LIN {X 0,Y 312.332,Z 608.768,A -85,B 0,C 180,E1 -15582.014,E2 -15582.014} C_VEL
LIN {X 0,Y 313.413,Z 600.363,A -85,B 0,C 180,E1 -15583.949,E2 -15583.949} C_VEL
LIN {X 0,Y 314.465,Z 591.676,A -85,B 0,C 180,E1 -15585.557,E2 -15585.557} C_VEL
LIN {X 0,Y 315.456,Z 582.123,A -85,B 0,C 180,E1 -15587.002,E2 -15587.002} C_VEL
LIN {X 0,Y 316.582,Z 571.707,A -85,B 0,C 180,E1 -15588.274,E2 -15588.274} C_VEL
LIN {X 0,Y 317.768,Z 560.291,A -85,B 0,C 180,E1 -15589.375,E2 -15589.375} C_VEL
LIN {X 0,Y 318.765,Z 548.571,A -85,B 0,C 180,E1 -15590.235,E2 -15590.235} C_VEL
LIN {X 0,Y 319.621,Z 535.041,A -85,B 0,C 180,E1 -15590.935,E2 -15590.935} C_VEL
LIN {X 0,Y 320.129,Z 521.595,A -85,B 0,C 180,E1 -15591.364,E2 -15591.364} C_VEL
LIN {X 0,Y 321.315,Z 456.274,A -85,B 0,C 180,E1 -15592.816,E2 -15592.816} C_VEL
LIN {X 0,Y 315.929,Z 420.388,A -85,B 0,C 180,E1 -15594.022,E2 -15594.022} C_VEL
LIN {X 0,Y 316.017,Z 418.253,A -85,B 0,C 180,E1 -15594.505,E2 -15594.505} C_VEL
LIN {X 0,Y 313.928,Z 406.505,A -85,B 0,C 180,E1 -15598.043,E2 -15598.043} C_VEL
LIN {X 0,Y 312.62,Z 400.101,A -85,B 0,C 180,E1 -15600.129,E2 -15600.129} C_VEL
LIN {X 0,Y 312.507,Z 400.053,A -85,B 0,C 180,E1 -15604.21,E2 -15604.21} C_VEL
LIN {X 0,Y 312.535,Z 400.049,A -85,B 0,C 180,E1 -15608.089,E2 -15608.089} C_VEL
LIN {X 0,Y 312.518,Z 400.054,A -85,B 0,C 180,E1 -15612.426,E2 -15612.426} C_VEL
LIN {X 0,Y 312.533,Z 400.041,A -85,B 0,C 180,E1 -15616.02,E2 -15616.02} C_VEL
LIN {X 0,Y 312.529,Z 400.055,A -85,B 0,C 180,E1 -15619.868,E2 -15619.868} C_VEL
LIN {X 0,Y 312.551,Z 400.049,A -85,B 0,C 180,E1 -15622.618,E2 -15622.618} C_VEL
LIN {X 0,Y 312.517,Z 400.054,A -85,B 0,C 180,E1 -15626.311,E2 -15626.311} C_VEL
LIN {X 0,Y 312.542,Z 400.047,A -85,B 0,C 180,E1 -15630.35,E2 -15630.35} C_VEL
LIN {X 0,Y 312.599,Z 400.044,A -85,B 0,C 180,E1 -15634.064,E2 -15634.064} C_VEL
LIN {X 0,Y 312.561,Z 400.049,A -85,B 0,C 180,E1 -15637.527,E2 -15637.527} C_VEL
LIN {X 0,Y 312.634,Z 400.04,A -85,B 0,C 180,E1 -15641.656,E2 -15641.656} C_VEL
LIN {X 0,Y 312.69,Z 400.034,A -85,B 0,C 180,E1 -15645.686,E2 -15645.686} C_VEL
LIN {X 0,Y 312.694,Z 400.027,A -85,B 0,C 180,E1 -15649.641,E2 -15649.641} C_VEL
LIN {X 0,Y 312.849,Z 400.01,A -85,B 0,C 180,E1 -15652.254,E2 -15652.254} C_VEL
LIN {X 0,Y 312.712,Z 400.031,A -85,B 0,C 180,E1 -15654.842,E2 -15654.842} C_VEL
LIN {X 0,Y 312.986,Z 399.993,A -85,B 0,C 180,E1 -15658.713,E2 -15658.713} C_VEL
LIN {X 0,Y 312.986,Z 399.99,A -85,B 0,C 180,E1 -15661.287,E2 -15661.287} C_VEL
LIN {X 0,Y 312.712,Z 400.032,A -85,B 0,C 180,E1 -15665.158,E2 -15665.158} C_VEL
LIN {X 0,Y 312.849,Z 400.013,A -85,B 0,C 180,E1 -15667.746,E2 -15667.746} C_VEL
LIN {X 0,Y 312.664,Z 400.027,A -85,B 0,C 180,E1 -15671.671,E2 -15671.671} C_VEL
LIN {X 0,Y 312.696,Z 400.029,A -85,B 0,C 180,E1 -15674.887,E2 -15674.887} C_VEL
LIN {X 0,Y 312.627,Z 400.044,A -85,B 0,C 180,E1 -15679.237,E2 -15679.237} C_VEL
LIN {X 0,Y 312.542,Z 400.047,A -85,B 0,C 180,E1 -15682.789,E2 -15682.789} C_VEL
LIN {X 0,Y 312.599,Z 400.041,A -85,B 0,C 180,E1 -15685.936,E2 -15685.936} C_VEL
LIN {X 0,Y 312.542,Z 400.051,A -85,B 0,C 180,E1 -15689.65,E2 -15689.65} C_VEL
LIN {X 0,Y 312.516,Z 400.048,A -85,B 0,C 180,E1 -15693.689,E2 -15693.689} C_VEL
LIN {X 0,Y 312.518,Z 400.057,A -85,B 0,C 180,E1 -15697.386,E2 -15697.386} C_VEL
LIN {X 0,Y 312.488,Z 400.058,A -85,B 0,C 180,E1 -15700.709,E2 -15700.709} C_VEL
LIN {X 0,Y 312.472,Z 400.058,A -85,B 0,C 180,E1 -15704.206,E2 -15704.206} C_VEL
LIN {X 0,Y 312.527,Z 400.05,A -85,B 0,C 180,E1 -15707.91,E2 -15707.91} C_VEL
LIN {X 0,Y 312.542,Z 400.052,A -85,B 0,C 180,E1 -15711.909,E2 -15711.909} C_VEL
LIN {X 0,Y 312.506,Z 400.048,A -85,B 0,C 180,E1 -15715.79,E2 -15715.79} C_VEL
LIN {X 0,Y 312.523,Z 400.047,A -85,B 0,C 180,E1 -15718.854,E2 -15718.854} C_VEL
LIN {X 0,Y 312.574,Z 400.047,A -85,B 0,C 180,E1 -15721.825,E2 -15721.825} C_VEL
LIN {X 0,Y 312.586,Z 400.042,A -85,B 0,C 180,E1 -15724.711,E2 -15724.711} C_VEL
LIN {X 0,Y 312.588,Z 400.047,A -85,B 0,C 180,E1 -15727.529,E2 -15727.529} C_VEL
LIN {X 0,Y 312.639,Z 400.028,A -85,B 0,C 180,E1 -15731.656,E2 -15731.656} C_VEL
LIN {X 0,Y 312.701,Z 400.206,A -85,B 0,C 180,E1 -15735.147,E2 -15735.147} C_VEL
LIN {X 0,Y 314.592,Z 410.211,A -85,B 0,C 180,E1 -15738.401,E2 -15738.401} C_VEL
LIN {X 0,Y 314.972,Z 412.171,A -85,B 0,C 180,E1 -15738.949,E2 -15738.949} C_VEL
LIN {X 0,Y 317.49,Z 420.363,A -85,B 0,C 180,E1 -15739.351,E2 -15739.351} C_VEL
LIN {X 0,Y 320.696,Z 439.395,A -85,B 0,C 180,E1 -15740.005,E2 -15740.005} C_VEL
LIN {X 0,Y 321.593,Z 445.108,A -85,B 0,C 180,E1 -15740.193,E2 -15740.193} C_VEL
LIN {X 0,Y 319.963,Z 519.638,A -85,B 0,C 180,E1 -15741.871,E2 -15741.871} C_VEL
LIN {X 0,Y 319.365,Z 532.672,A -85,B 0,C 180,E1 -15742.413,E2 -15742.413} C_VEL
LIN {X 0,Y 318.56,Z 545.103,A -85,B 0,C 180,E1 -15743.177,E2 -15743.177} C_VEL
LIN {X 0,Y 317.505,Z 556.543,A -85,B 0,C 180,E1 -15744.124,E2 -15744.124} C_VEL
LIN {X 0,Y 316.221,Z 568.185,A -85,B 0,C 180,E1 -15745.379,E2 -15745.379} C_VEL
LIN {X 0,Y 314.984,Z 578.646,A -85,B 0,C 180,E1 -15746.802,E2 -15746.802} C_VEL
LIN {X 0,Y 313.883,Z 588.052,A -85,B 0,C 180,E1 -15748.396,E2 -15748.396} C_VEL
LIN {X 0,Y 312.774,Z 597.128,A -85,B 0,C 180,E1 -15750.322,E2 -15750.322} C_VEL
LIN {X 0,Y 312.008,Z 604.437,A -85,B 0,C 180,E1 -15752.259,E2 -15752.259} C_VEL
LIN {X 0,Y 311.384,Z 609.404,A -85,B 0,C 180,E1 -15753.882,E2 -15753.882} C_VEL
LIN {X 0,Y 311.069,Z 614.19,A -85,B 0,C 180,E1 -15755.827,E2 -15755.827} C_VEL
LIN {X 0,Y 310.787,Z 617.906,A -85,B 0,C 180,E1 -15757.798,E2 -15757.798} C_VEL
LIN {X 0,Y 310.591,Z 619.823,A -85,B 0,C 180,E1 -15759.113,E2 -15759.113} C_VEL
LIN {X 0,Y 310.484,Z 621.266,A -85,B 0,C 180,E1 -15760.432,E2 -15760.432} C_VEL
LIN {X 0,Y 310.487,Z 622.287,A -85,B 0,C 180,E1 -15761.754,E2 -15761.754} C_VEL
LIN {X 0,Y 310.52,Z 622.988,A -85,B 0,C 180,E1 -15763.29,E2 -15763.29} C_VEL
LIN {X 0,Y 310.477,Z 622.899,A -85,B 0,C 180,E1 -15765.761,E2 -15765.761} C_VEL
LIN {X 0,Y 310.849,Z 621.362,A -85,B 0,C 180,E1 -15768.272,E2 -15768.272} C_VEL
LIN {X 0,Y 311.123,Z 619.69,A -85,B 0,C 180,E1 -15769.805,E2 -15769.805} C_VEL
LIN {X 0,Y 311.721,Z 616.547,A -85,B 0,C 180,E1 -15771.839,E2 -15771.839} C_VEL
LIN {X 0,Y 312.536,Z 612.255,A -85,B 0,C 180,E1 -15773.876,E2 -15773.876} C_VEL
LIN {X 0,Y 313.634,Z 606.844,A -85,B 0,C 180,E1 -15775.854,E2 -15775.854} C_VEL
LIN {X 0,Y 315.1,Z 599.633,A -85,B 0,C 180,E1 -15777.929,E2 -15777.929} C_VEL
LIN {X 0,Y 316.754,Z 591.555,A -85,B 0,C 180,E1 -15779.771,E2 -15779.771} C_VEL
LIN {X 0,Y 318.433,Z 582.51,A -85,B 0,C 180,E1 -15781.426,E2 -15781.426} C_VEL
LIN {X 0,Y 320.298,Z 572.505,A -85,B 0,C 180,E1 -15782.891,E2 -15782.891} C_VEL
LIN {X 0,Y 321.96,Z 561.76,A -85,B 0,C 180,E1 -15784.159,E2 -15784.159} C_VEL
LIN {X 0,Y 323.509,Z 549.927,A -85,B 0,C 180,E1 -15785.242,E2 -15785.242} C_VEL
LIN {X 0,Y 324.743,Z 538.352,A -85,B 0,C 180,E1 -15786.041,E2 -15786.041} C_VEL
LIN {X 0,Y 325.821,Z 525.426,A -85,B 0,C 180,E1 -15786.67,E2 -15786.67} C_VEL
LIN {X 0,Y 326.468,Z 511.967,A -85,B 0,C 180,E1 -15787.067,E2 -15787.067} C_VEL
LIN {X 0,Y 328.157,Z 446.992,A -85,B 0,C 180,E1 -15788.521,E2 -15788.521} C_VEL
LIN {X 0,Y 325.249,Z 434.051,A -85,B 0,C 180,E1 -15789.147,E2 -15789.147} C_VEL
LIN {X 0,Y 321.952,Z 426.371,A -85,B 0,C 180,E1 -15789.693,E2 -15789.693} C_VEL
LIN {X 0,Y 319.927,Z 423.383,A -85,B 0,C 180,E1 -15789.995,E2 -15789.995} C_VEL
LIN {X 0,Y 315.274,Z 419.81,A -85,B 0,C 180,E1 -15790.605,E2 -15790.605} C_VEL
LIN {X 0,Y 310.624,Z 416.297,A -85,B 0,C 180,E1 -15791.239,E2 -15791.239} C_VEL
LIN {X 0,Y 308.623,Z 413.402,A -85,B 0,C 180,E1 -15791.58,E2 -15791.58} C_VEL
LIN {X 0,Y 308.228,Z 412.248,A -85,B 0,C 180,E1 -15791.753,E2 -15791.753} C_VEL
LIN {X 0,Y 306.422,Z 404.582,A -85,B 0,C 180,E1 -15794.683,E2 -15794.683} C_VEL
LIN {X 0,Y 305.53,Z 400.961,A -85,B 0,C 180,E1 -15796.243,E2 -15796.243} C_VEL
LIN {X 0,Y 305.48,Z 400.933,A -85,B 0,C 180,E1 -15799.896,E2 -15799.896} C_VEL
LIN {X 0,Y 305.496,Z 400.931,A -85,B 0,C 180,E1 -15803.626,E2 -15803.626} C_VEL
LIN {X 0,Y 305.46,Z 400.927,A -85,B 0,C 180,E1 -15806.483,E2 -15806.483} C_VEL
LIN {X 0,Y 305.46,Z 400.916,A -85,B 0,C 180,E1 -15809.591,E2 -15809.591} C_VEL
LIN {X 0,Y 305.528,Z 400.927,A -85,B 0,C 180,E1 -15812.609,E2 -15812.609} C_VEL
LIN {X 0,Y 305.502,Z 400.93,A -85,B 0,C 180,E1 -15815.538,E2 -15815.538} C_VEL
LIN {X 0,Y 305.524,Z 400.927,A -85,B 0,C 180,E1 -15819.815,E2 -15819.815} C_VEL
LIN {X 0,Y 305.568,Z 400.918,A -85,B 0,C 180,E1 -15822.603,E2 -15822.603} C_VEL
LIN {X 0,Y 305.642,Z 400.904,A -85,B 0,C 180,E1 -15825.349,E2 -15825.349} C_VEL
LIN {X 0,Y 305.633,Z 400.903,A -85,B 0,C 180,E1 -15829.4,E2 -15829.4} C_VEL
LIN {X 0,Y 305.805,Z 400.892,A -85,B 0,C 180,E1 -15832.074,E2 -15832.074} C_VEL
LIN {X 0,Y 305.686,Z 400.897,A -85,B 0,C 180,E1 -15834.724,E2 -15834.724} C_VEL
LIN {X 0,Y 305.955,Z 400.864,A -85,B 0,C 180,E1 -15838.684,E2 -15838.684} C_VEL
LIN {X 0,Y 305.954,Z 400.874,A -85,B 0,C 180,E1 -15841.316,E2 -15841.316} C_VEL
LIN {X 0,Y 305.684,Z 400.905,A -85,B 0,C 180,E1 -15845.277,E2 -15845.277} C_VEL
LIN {X 0,Y 305.805,Z 400.886,A -85,B 0,C 180,E1 -15847.926,E2 -15847.926} C_VEL
LIN {X 0,Y 305.599,Z 400.917,A -85,B 0,C 180,E1 -15851.945,E2 -15851.945} C_VEL
LIN {X 0,Y 305.631,Z 400.911,A -85,B 0,C 180,E1 -15855.035,E2 -15855.035} C_VEL
LIN {X 0,Y 305.57,Z 400.919,A -85,B 0,C 180,E1 -15859.446,E2 -15859.446} C_VEL
LIN {X 0,Y 305.484,Z 400.924,A -85,B 0,C 180,E1 -15863.042,E2 -15863.042} C_VEL
LIN {X 0,Y 305.541,Z 400.919,A -85,B 0,C 180,E1 -15866.228,E2 -15866.228} C_VEL
LIN {X 0,Y 305.49,Z 400.931,A -85,B 0,C 180,E1 -15869.051,E2 -15869.051} C_VEL
LIN {X 0,Y 305.46,Z 400.932,A -85,B 0,C 180,E1 -15873.518,E2 -15873.518} C_VEL
LIN {X 0,Y 305.498,Z 400.927,A -85,B 0,C 180,E1 -15876.736,E2 -15876.736} C_VEL
LIN {X 0,Y 305.49,Z 400.914,A -85,B 0,C 180,E1 -15880.609,E2 -15880.609} C_VEL
LIN {X 0,Y 305.489,Z 400.932,A -85,B 0,C 180,E1 -15883.644,E2 -15883.644} C_VEL
LIN {X 0,Y 305.48,Z 400.925,A -85,B 0,C 180,E1 -15887.41,E2 -15887.41} C_VEL
LIN {X 0,Y 305.493,Z 400.932,A -85,B 0,C 180,E1 -15891.602,E2 -15891.602} C_VEL
LIN {X 0,Y 305.498,Z 401.029,A -85,B 0,C 180,E1 -15894.691,E2 -15894.691} C_VEL
LIN {X 0,Y 307.861,Z 410.376,A -85,B 0,C 180,E1 -15898.329,E2 -15898.329} C_VEL
LIN {X 0,Y 309.922,Z 419.562,A -85,B 0,C 180,E1 -15901.563,E2 -15901.563} C_VEL
LIN {X 0,Y 313.421,Z 427.22,A -85,B 0,C 180,E1 -15902.233,E2 -15902.233} C_VEL
LIN {X 0,Y 316.75,Z 435.265,A -85,B 0,C 180,E1 -15902.823,E2 -15902.823} C_VEL
LIN {X 0,Y 320.789,Z 454.521,A -85,B 0,C 180,E1 -15903.763,E2 -15903.763} C_VEL
LIN {X 0,Y 321.79,Z 460.542,A -85,B 0,C 180,E1 -15904.023,E2 -15904.023} C_VEL
LIN {X 0,Y 319.782,Z 527.928,A -85,B 0,C 180,E1 -15905.579,E2 -15905.579} C_VEL
LIN {X 0,Y 318.81,Z 540.907,A -85,B 0,C 180,E1 -15906.106,E2 -15906.106} C_VEL
LIN {X 0,Y 317.437,Z 553.468,A -85,B 0,C 180,E1 -15906.861,E2 -15906.861} C_VEL
LIN {X 0,Y 316.006,Z 564.655,A -85,B 0,C 180,E1 -15907.786,E2 -15907.786} C_VEL
LIN {X 0,Y 314.12,Z 576.238,A -85,B 0,C 180,E1 -15909.025,E2 -15909.025} C_VEL
LIN {X 0,Y 312.255,Z 586.659,A -85,B 0,C 180,E1 -15910.441,E2 -15910.441} C_VEL
LIN {X 0,Y 310.511,Z 595.458,A -85,B 0,C 180,E1 -15911.919,E2 -15911.919} C_VEL
LIN {X 0,Y 308.774,Z 604.486,A -85,B 0,C 180,E1 -15913.811,E2 -15913.811} C_VEL
LIN {X 0,Y 307.072,Z 611.943,A -85,B 0,C 180,E1 -15915.758,E2 -15915.758} C_VEL
LIN {X 0,Y 305.684,Z 618.85,A -85,B 0,C 180,E1 -15918.059,E2 -15918.059} C_VEL
LIN {X 0,Y 304.772,Z 623.43,A -85,B 0,C 180,E1 -15920.041,E2 -15920.041} C_VEL
LIN {X 0,Y 304.128,Z 626.927,A -85,B 0,C 180,E1 -15922.031,E2 -15922.031} C_VEL
LIN {X 0,Y 303.783,Z 629.584,A -85,B 0,C 180,E1 -15924.159,E2 -15924.159} C_VEL
LIN {X 0,Y 303.608,Z 631.026,A -85,B 0,C 180,E1 -15926.018,E2 -15926.018} C_VEL
LIN {X 0,Y 303.582,Z 631.609,A -85,B 0,C 180,E1 -15927.347,E2 -15927.347} C_VEL
LIN {X 0,Y 303.528,Z 631.779,A -85,B 0,C 180,E1 -15928.674,E2 -15928.674} C_VEL
LIN {X 0,Y 303.545,Z 631.537,A -85,B 0,C 180,E1 -15930,E2 -15930} C_VEL
LIN {X 0,Y 303.58,Z 629.892,A -85,B 0,C 180,E1 -15932.654,E2 -15932.654} C_VEL
LIN {X 0,Y 303.584,Z 628.446,A -85,B 0,C 180,E1 -15933.983,E2 -15933.983} C_VEL
LIN {X 0,Y 303.618,Z 626.19,A -85,B 0,C 180,E1 -15935.53,E2 -15935.53} C_VEL
LIN {X 0,Y 303.995,Z 621.397,A -85,B 0,C 180,E1 -15937.974,E2 -15937.974} C_VEL
LIN {X 0,Y 304.608,Z 615.141,A -85,B 0,C 180,E1 -15940.301,E2 -15940.301} C_VEL
LIN {X 0,Y 305.353,Z 608.311,A -85,B 0,C 180,E1 -15942.292,E2 -15942.292} C_VEL
LIN {X 0,Y 306.473,Z 599.799,A -85,B 0,C 180,E1 -15944.272,E2 -15944.272} C_VEL
LIN {X 0,Y 307.726,Z 589.82,A -85,B 0,C 180,E1 -15946.111,E2 -15946.111} C_VEL
LIN {X 0,Y 308.901,Z 578.948,A -85,B 0,C 180,E1 -15947.716,E2 -15947.716} C_VEL
LIN {X 0,Y 310.122,Z 567.713,A -85,B 0,C 180,E1 -15949.012,E2 -15949.012} C_VEL
LIN {X 0,Y 311.398,Z 555.107,A -85,B 0,C 180,E1 -15950.132,E2 -15950.132} C_VEL
LIN {X 0,Y 312.406,Z 542.157,A -85,B 0,C 180,E1 -15950.967,E2 -15950.967} C_VEL
LIN {X 0,Y 313.17,Z 528.284,A -85,B 0,C 180,E1 -15951.56,E2 -15951.56} C_VEL
LIN {X 0,Y 314.635,Z 457.597,A -85,B 0,C 180,E1 -15953.196,E2 -15953.196} C_VEL
LIN {X 0,Y 309.07,Z 420.436,A -85,B 0,C 180,E1 -15954.474,E2 -15954.474} C_VEL
LIN {X 0,Y 309.035,Z 419.339,A -85,B 0,C 180,E1 -15954.659,E2 -15954.659} C_VEL
LIN {X 0,Y 307.124,Z 408.508,A -85,B 0,C 180,E1 -15957.976,E2 -15957.976} C_VEL
LIN {X 0,Y 305.525,Z 401.019,A -85,B 0,C 180,E1 -15960.45,E2 -15960.45} C_VEL
LIN {X 0,Y 305.465,Z 400.931,A -85,B 0,C 180,E1 -15964.078,E2 -15964.078} C_VEL
LIN {X 0,Y 305.496,Z 400.93,A -85,B 0,C 180,E1 -15966.736,E2 -15966.736} C_VEL
LIN {X 0,Y 305.454,Z 400.933,A -85,B 0,C 180,E1 -15970.599,E2 -15970.599} C_VEL
LIN {X 0,Y 305.452,Z 400.931,A -85,B 0,C 180,E1 -15973.65,E2 -15973.65} C_VEL
LIN {X 0,Y 305.506,Z 400.918,A -85,B 0,C 180,E1 -15977.403,E2 -15977.403} C_VEL
LIN {X 0,Y 305.518,Z 400.929,A -85,B 0,C 180,E1 -15981.604,E2 -15981.604} C_VEL
LIN {X 0,Y 305.46,Z 400.93,A -85,B 0,C 180,E1 -15984.886,E2 -15984.886} C_VEL
LIN {X 0,Y 305.449,Z 400.935,A -85,B 0,C 180,E1 -15988.355,E2 -15988.355} C_VEL
LIN {X 0,Y 305.518,Z 400.924,A -85,B 0,C 180,E1 -15991.113,E2 -15991.113} C_VEL
LIN {X 0,Y 305.568,Z 400.92,A -85,B 0,C 180,E1 -15994.087,E2 -15994.087} C_VEL
LIN {X 0,Y 305.478,Z 400.926,A -85,B 0,C 180,E1 -15998.401,E2 -15998.401} C_VEL
LIN {X 0,Y 305.576,Z 400.915,A -85,B 0,C 180,E1 -16001.217,E2 -16001.217} C_VEL
LIN {X 0,Y 305.645,Z 400.914,A -85,B 0,C 180,E1 -16005.349,E2 -16005.349} C_VEL
LIN {X 0,Y 305.631,Z 400.905,A -85,B 0,C 180,E1 -16009.399,E2 -16009.399} C_VEL
LIN {X 0,Y 305.793,Z 400.889,A -85,B 0,C 180,E1 -16012.074,E2 -16012.074} C_VEL
LIN {X 0,Y 305.683,Z 400.906,A -85,B 0,C 180,E1 -16014.723,E2 -16014.723} C_VEL
LIN {X 0,Y 305.953,Z 400.869,A -85,B 0,C 180,E1 -16018.684,E2 -16018.684} C_VEL
LIN {X 0,Y 305.953,Z 400.865,A -85,B 0,C 180,E1 -16021.316,E2 -16021.316} C_VEL
LIN {X 0,Y 305.683,Z 400.909,A -85,B 0,C 180,E1 -16025.277,E2 -16025.277} C_VEL
LIN {X 0,Y 305.793,Z 400.891,A -85,B 0,C 180,E1 -16027.926,E2 -16027.926} C_VEL
LIN {X 0,Y 305.598,Z 400.905,A -85,B 0,C 180,E1 -16031.945,E2 -16031.945} C_VEL
LIN {X 0,Y 305.634,Z 400.909,A -85,B 0,C 180,E1 -16035.035,E2 -16035.035} C_VEL
LIN {X 0,Y 305.573,Z 400.92,A -85,B 0,C 180,E1 -16039.445,E2 -16039.445} C_VEL
LIN {X 0,Y 305.487,Z 400.924,A -85,B 0,C 180,E1 -16043.041,E2 -16043.041} C_VEL
LIN {X 0,Y 305.544,Z 400.919,A -85,B 0,C 180,E1 -16046.227,E2 -16046.227} C_VEL
LIN {X 0,Y 305.493,Z 400.933,A -85,B 0,C 180,E1 -16049.05,E2 -16049.05} C_VEL
LIN {X 0,Y 305.462,Z 400.927,A -85,B 0,C 180,E1 -16053.517,E2 -16053.517} C_VEL
LIN {X 0,Y 305.47,Z 400.932,A -85,B 0,C 180,E1 -16056.74,E2 -16056.74} C_VEL
LIN {X 0,Y 305.452,Z 400.933,A -85,B 0,C 180,E1 -16060.6,E2 -16060.6} C_VEL
LIN {X 0,Y 305.423,Z 400.937,A -85,B 0,C 180,E1 -16064.494,E2 -16064.494} C_VEL
LIN {X 0,Y 305.475,Z 400.929,A -85,B 0,C 180,E1 -16068.15,E2 -16068.15} C_VEL
LIN {X 0,Y 305.507,Z 400.929,A -85,B 0,C 180,E1 -16071.603,E2 -16071.603} C_VEL
LIN {X 0,Y 305.462,Z 400.931,A -85,B 0,C 180,E1 -16074.887,E2 -16074.887} C_VEL
LIN {X 0,Y 305.451,Z 400.923,A -85,B 0,C 180,E1 -16078.355,E2 -16078.355} C_VEL
LIN {X 0,Y 305.52,Z 400.93,A -85,B 0,C 180,E1 -16081.114,E2 -16081.114} C_VEL
LIN {X 0,Y 305.566,Z 400.915,A -85,B 0,C 180,E1 -16084.088,E2 -16084.088} C_VEL
LIN {X 0,Y 305.502,Z 400.93,A -85,B 0,C 180,E1 -16088.403,E2 -16088.403} C_VEL
LIN {X 0,Y 305.591,Z 400.904,A -85,B 0,C 180,E1 -16091.218,E2 -16091.218} C_VEL
LIN {X 0,Y 305.658,Z 401.072,A -85,B 0,C 180,E1 -16094.813,E2 -16094.813} C_VEL
LIN {X 0,Y 307.557,Z 411.003,A -85,B 0,C 180,E1 -16098.132,E2 -16098.132} C_VEL
LIN {X 0,Y 307.829,Z 412.394,A -85,B 0,C 180,E1 -16098.479,E2 -16098.479} C_VEL
LIN {X 0,Y 310.923,Z 422.04,A -85,B 0,C 180,E1 -16098.96,E2 -16098.96} C_VEL
LIN {X 0,Y 314.103,Z 440.853,A -85,B 0,C 180,E1 -16099.623,E2 -16099.623} C_VEL
LIN {X 0,Y 314.893,Z 446.011,A -85,B 0,C 180,E1 -16099.797,E2 -16099.797} C_VEL
LIN {X 0,Y 313.253,Z 518.575,A -85,B 0,C 180,E1 -16101.452,E2 -16101.452} C_VEL
LIN {X 0,Y 312.698,Z 531.262,A -85,B 0,C 180,E1 -16101.965,E2 -16101.965} C_VEL
LIN {X 0,Y 311.83,Z 544.047,A -85,B 0,C 180,E1 -16102.741,E2 -16102.741} C_VEL
LIN {X 0,Y 310.79,Z 555.378,A -85,B 0,C 180,E1 -16103.671,E2 -16103.671} C_VEL
LIN {X 0,Y 309.594,Z 566.023,A -85,B 0,C 180,E1 -16104.79,E2 -16104.79} C_VEL
LIN {X 0,Y 308.478,Z 575.797,A -85,B 0,C 180,E1 -16106.081,E2 -16106.081} C_VEL
LIN {X 0,Y 307.176,Z 585.738,A -85,B 0,C 180,E1 -16107.705,E2 -16107.705} C_VEL
LIN {X 0,Y 306.254,Z 593.861,A -85,B 0,C 180,E1 -16109.342,E2 -16109.342} C_VEL
LIN {X 0,Y 305.197,Z 601.864,A -85,B 0,C 180,E1 -16111.319,E2 -16111.319} C_VEL
LIN {X 0,Y 304.475,Z 608.254,A -85,B 0,C 180,E1 -16113.308,E2 -16113.308} C_VEL
LIN {X 0,Y 304.063,Z 613.325,A -85,B 0,C 180,E1 -16115.304,E2 -16115.304} C_VEL
LIN {X 0,Y 303.777,Z 617.265,A -85,B 0,C 180,E1 -16117.31,E2 -16117.31} C_VEL
LIN {X 0,Y 303.473,Z 620.176,A -85,B 0,C 180,E1 -16119.329,E2 -16119.329} C_VEL
LIN {X 0,Y 303.384,Z 621.548,A -85,B 0,C 180,E1 -16120.679,E2 -16120.679} C_VEL
LIN {X 0,Y 303.383,Z 622.518,A -85,B 0,C 180,E1 -16122.033,E2 -16122.033} C_VEL
LIN {X 0,Y 303.427,Z 623.09,A -85,B 0,C 180,E1 -16123.392,E2 -16123.392} C_VEL
LIN {X 0,Y 303.361,Z 623.213,A -85,B 0,C 180,E1 -16124.763,E2 -16124.763} C_VEL
LIN {X 0,Y 303.408,Z 622.923,A -85,B 0,C 180,E1 -16126.138,E2 -16126.138} C_VEL
LIN {X 0,Y 303.81,Z 621.473,A -85,B 0,C 180,E1 -16128.478,E2 -16128.478} C_VEL
LIN {X 0,Y 304.357,Z 618.557,A -85,B 0,C 180,E1 -16130.971,E2 -16130.971} C_VEL
LIN {X 0,Y 305.095,Z 614.922,A -85,B 0,C 180,E1 -16133.053,E2 -16133.053} C_VEL
LIN {X 0,Y 306.123,Z 610.082,A -85,B 0,C 180,E1 -16135.132,E2 -16135.132} C_VEL
LIN {X 0,Y 307.444,Z 603.879,A -85,B 0,C 180,E1 -16137.205,E2 -16137.205} C_VEL
LIN {X 0,Y 309.108,Z 596.084,A -85,B 0,C 180,E1 -16139.263,E2 -16139.263} C_VEL
LIN {X 0,Y 310.946,Z 587.398,A -85,B 0,C 180,E1 -16141.079,E2 -16141.079} C_VEL
LIN {X 0,Y 312.756,Z 578.142,A -85,B 0,C 180,E1 -16142.635,E2 -16142.635} C_VEL
LIN {X 0,Y 314.492,Z 568.389,A -85,B 0,C 180,E1 -16143.963,E2 -16143.963} C_VEL
LIN {X 0,Y 316.152,Z 557.714,A -85,B 0,C 180,E1 -16145.129,E2 -16145.129} C_VEL
LIN {X 0,Y 317.704,Z 545.272,A -85,B 0,C 180,E1 -16146.181,E2 -16146.181} C_VEL
LIN {X 0,Y 319.049,Z 532.166,A -85,B 0,C 180,E1 -16146.968,E2 -16146.968} C_VEL
LIN {X 0,Y 319.913,Z 519.714,A -85,B 0,C 180,E1 -16147.471,E2 -16147.471} C_VEL
LIN {X 0,Y 322.056,Z 448.446,A -85,B 0,C 180,E1 -16149.111,E2 -16149.111} C_VEL
LIN {X 0,Y 319.404,Z 436.749,A -85,B 0,C 180,E1 -16149.698,E2 -16149.698} C_VEL
LIN {X 0,Y 312.065,Z 420.297,A -85,B 0,C 180,E1 -16150.961,E2 -16150.961} C_VEL
LIN {X 0,Y 308.623,Z 413.402,A -85,B 0,C 180,E1 -16151.58,E2 -16151.58} C_VEL
LIN {X 0,Y 307.63,Z 412.085,A -85,B 0,C 180,E1 -16151.882,E2 -16151.882} C_VEL
LIN {X 0,Y 302.646,Z 408.369,A -85,B 0,C 180,E1 -16153.836,E2 -16153.836} C_VEL
LIN {X 0,Y 300.585,Z 406.45,A -85,B 0,C 180,E1 -16154.954,E2 -16154.954} C_VEL
LIN {X 0,Y 299.117,Z 403.891,A -85,B 0,C 180,E1 -16156.07,E2 -16156.07} C_VEL
LIN {X 0,Y 298.534,Z 402.112,A -85,B 0,C 180,E1 -16156.826,E2 -16156.826} C_VEL
LIN {X 0,Y 298.47,Z 401.799,A -85,B 0,C 180,E1 -16157.393,E2 -16157.393} C_VEL
LIN {X 0,Y 298.431,Z 401.8,A -85,B 0,C 180,E1 -16160.998,E2 -16160.998} C_VEL
LIN {X 0,Y 298.428,Z 401.807,A -85,B 0,C 180,E1 -16163.932,E2 -16163.932} C_VEL
LIN {X 0,Y 298.394,Z 401.816,A -85,B 0,C 180,E1 -16167.981,E2 -16167.981} C_VEL
LIN {X 0,Y 298.464,Z 401.799,A -85,B 0,C 180,E1 -16171.904,E2 -16171.904} C_VEL
LIN {X 0,Y 298.48,Z 401.801,A -85,B 0,C 180,E1 -16174.924,E2 -16174.924} C_VEL
LIN {X 0,Y 298.451,Z 401.81,A -85,B 0,C 180,E1 -16179.315,E2 -16179.315} C_VEL
LIN {X 0,Y 298.532,Z 401.792,A -85,B 0,C 180,E1 -16182.179,E2 -16182.179} C_VEL
LIN {X 0,Y 298.586,Z 401.784,A -85,B 0,C 180,E1 -16184.994,E2 -16184.994} C_VEL
LIN {X 0,Y 298.588,Z 401.782,A -85,B 0,C 180,E1 -16189.147,E2 -16189.147} C_VEL
LIN {X 0,Y 298.751,Z 401.771,A -85,B 0,C 180,E1 -16191.886,E2 -16191.886} C_VEL
LIN {X 0,Y 298.657,Z 401.772,A -85,B 0,C 180,E1 -16194.599,E2 -16194.599} C_VEL
LIN {X 0,Y 298.922,Z 401.74,A -85,B 0,C 180,E1 -16198.653,E2 -16198.653} C_VEL
LIN {X 0,Y 298.92,Z 401.75,A -85,B 0,C 180,E1 -16201.347,E2 -16201.347} C_VEL
LIN {X 0,Y 298.654,Z 401.782,A -85,B 0,C 180,E1 -16205.401,E2 -16205.401} C_VEL
LIN {X 0,Y 298.751,Z 401.763,A -85,B 0,C 180,E1 -16208.114,E2 -16208.114} C_VEL
LIN {X 0,Y 298.549,Z 401.794,A -85,B 0,C 180,E1 -16212.232,E2 -16212.232} C_VEL
LIN {X 0,Y 298.599,Z 401.79,A -85,B 0,C 180,E1 -16215.21,E2 -16215.21} C_VEL
LIN {X 0,Y 298.533,Z 401.793,A -85,B 0,C 180,E1 -16219.244,E2 -16219.244} C_VEL
LIN {X 0,Y 298.451,Z 401.804,A -85,B 0,C 180,E1 -16223.598,E2 -16223.598} C_VEL
LIN {X 0,Y 298.484,Z 401.797,A -85,B 0,C 180,E1 -16226.575,E2 -16226.575} C_VEL
LIN {X 0,Y 298.415,Z 401.811,A -85,B 0,C 180,E1 -16229.642,E2 -16229.642} C_VEL
LIN {X 0,Y 298.39,Z 401.816,A -85,B 0,C 180,E1 -16232.801,E2 -16232.801} C_VEL
LIN {X 0,Y 298.466,Z 401.803,A -85,B 0,C 180,E1 -16236.815,E2 -16236.815} C_VEL
LIN {X 0,Y 298.451,Z 401.787,A -85,B 0,C 180,E1 -16241.104,E2 -16241.104} C_VEL
LIN {X 0,Y 298.456,Z 401.799,A -85,B 0,C 180,E1 -16243.117,E2 -16243.117} C_VEL
LIN {X 0,Y 298.429,Z 401.798,A -85,B 0,C 180,E1 -16246.927,E2 -16246.927} C_VEL
LIN {X 0,Y 298.413,Z 401.805,A -85,B 0,C 180,E1 -16251.004,E2 -16251.004} C_VEL
LIN {X 0,Y 298.476,Z 401.931,A -85,B 0,C 180,E1 -16253.94,E2 -16253.94} C_VEL
LIN {X 0,Y 300.951,Z 411.844,A -85,B 0,C 180,E1 -16257.91,E2 -16257.91} C_VEL
LIN {X 0,Y 302.785,Z 419.699,A -85,B 0,C 180,E1 -16260.718,E2 -16260.718} C_VEL
LIN {X 0,Y 309.659,Z 434.591,A -85,B 0,C 180,E1 -16261.997,E2 -16261.997} C_VEL
LIN {X 0,Y 311.216,Z 438.905,A -85,B 0,C 180,E1 -16262.295,E2 -16262.295} C_VEL
LIN {X 0,Y 315.03,Z 457.761,A -85,B 0,C 180,E1 -16263.229,E2 -16263.229} C_VEL
LIN {X 0,Y 315.631,Z 462.344,A -85,B 0,C 180,E1 -16263.416,E2 -16263.416} C_VEL
LIN {X 0,Y 313.536,Z 528.292,A -85,B 0,C 180,E1 -16264.971,E2 -16264.971} C_VEL
LIN {X 0,Y 312.471,Z 541.867,A -85,B 0,C 180,E1 -16265.545,E2 -16265.545} C_VEL
LIN {X 0,Y 310.991,Z 554.637,A -85,B 0,C 180,E1 -16266.352,E2 -16266.352} C_VEL
LIN {X 0,Y 309.502,Z 565.504,A -85,B 0,C 180,E1 -16267.293,E2 -16267.293} C_VEL
LIN {X 0,Y 307.552,Z 576.909,A -85,B 0,C 180,E1 -16268.555,E2 -16268.555} C_VEL
LIN {X 0,Y 305.597,Z 587.201,A -85,B 0,C 180,E1 -16269.997,E2 -16269.997} C_VEL
LIN {X 0,Y 303.707,Z 596.291,A -85,B 0,C 180,E1 -16271.582,E2 -16271.582} C_VEL
LIN {X 0,Y 301.967,Z 604.788,A -85,B 0,C 180,E1 -16273.435,E2 -16273.435} C_VEL
LIN {X 0,Y 300.207,Z 612.17,A -85,B 0,C 180,E1 -16275.425,E2 -16275.425} C_VEL
LIN {X 0,Y 298.726,Z 619,A -85,B 0,C 180,E1 -16277.776,E2 -16277.776} C_VEL
LIN {X 0,Y 297.779,Z 623.521,A -85,B 0,C 180,E1 -16279.805,E2 -16279.805} C_VEL
LIN {X 0,Y 297.082,Z 626.975,A -85,B 0,C 180,E1 -16281.84,E2 -16281.84} C_VEL
LIN {X 0,Y 296.621,Z 630.041,A -85,B 0,C 180,E1 -16284.562,E2 -16284.562} C_VEL
LIN {X 0,Y 296.488,Z 631.539,A -85,B 0,C 180,E1 -16287.283,E2 -16287.283} C_VEL
LIN {X 0,Y 296.45,Z 631.667,A -85,B 0,C 180,E1 -16288.642,E2 -16288.642} C_VEL
LIN {X 0,Y 296.462,Z 631.402,A -85,B 0,C 180,E1 -16290,E2 -16290} C_VEL
LIN {X 0,Y 296.45,Z 630.751,A -85,B 0,C 180,E1 -16291.359,E2 -16291.359} C_VEL
LIN {X 0,Y 296.485,Z 629.71,A -85,B 0,C 180,E1 -16292.718,E2 -16292.718} C_VEL
LIN {X 0,Y 296.485,Z 628.216,A -85,B 0,C 180,E1 -16294.078,E2 -16294.078} C_VEL
LIN {X 0,Y 296.572,Z 625.175,A -85,B 0,C 180,E1 -16296.121,E2 -16296.121} C_VEL
LIN {X 0,Y 296.93,Z 621.065,A -85,B 0,C 180,E1 -16298.165,E2 -16298.165} C_VEL
LIN {X 0,Y 297.58,Z 614.748,A -85,B 0,C 180,E1 -16300.547,E2 -16300.547} C_VEL
LIN {X 0,Y 298.358,Z 607.852,A -85,B 0,C 180,E1 -16302.585,E2 -16302.585} C_VEL
LIN {X 0,Y 299.358,Z 600.808,A -85,B 0,C 180,E1 -16304.271,E2 -16304.271} C_VEL
LIN {X 0,Y 300.469,Z 592.301,A -85,B 0,C 180,E1 -16305.952,E2 -16305.952} C_VEL
LIN {X 0,Y 301.44,Z 583.665,A -85,B 0,C 180,E1 -16307.358,E2 -16307.358} C_VEL
LIN {X 0,Y 302.7,Z 572.73,A -85,B 0,C 180,E1 -16308.793,E2 -16308.793} C_VEL
LIN {X 0,Y 303.939,Z 561.604,A -85,B 0,C 180,E1 -16309.942,E2 -16309.942} C_VEL
LIN {X 0,Y 305.104,Z 549.245,A -85,B 0,C 180,E1 -16310.918,E2 -16310.918} C_VEL
LIN {X 0,Y 305.991,Z 536.125,A -85,B 0,C 180,E1 -16311.649,E2 -16311.649} C_VEL
LIN {X 0,Y 306.572,Z 523.57,A -85,B 0,C 180,E1 -16312.092,E2 -16312.092} C_VEL
LIN {X 0,Y 307.827,Z 457.354,A -85,B 0,C 180,E1 -16313.638,E2 -16313.638} C_VEL
LIN {X 0,Y 302.332,Z 421.313,A -85,B 0,C 180,E1 -16314.906,E2 -16314.906} C_VEL
LIN {X 0,Y 301.956,Z 419.714,A -85,B 0,C 180,E1 -16315.053,E2 -16315.053} C_VEL
LIN {X 0,Y 300.031,Z 409.244,A -85,B 0,C 180,E1 -16318.316,E2 -16318.316} C_VEL
LIN {X 0,Y 298.483,Z 401.893,A -85,B 0,C 180,E1 -16320.804,E2 -16320.804} C_VEL
LIN {X 0,Y 298.428,Z 401.806,A -85,B 0,C 180,E1 -16324.487,E2 -16324.487} C_VEL
LIN {X 0,Y 298.432,Z 401.807,A -85,B 0,C 180,E1 -16327.755,E2 -16327.755} C_VEL
LIN {X 0,Y 298.413,Z 401.813,A -85,B 0,C 180,E1 -16331.256,E2 -16331.256} C_VEL
LIN {X 0,Y 298.416,Z 401.8,A -85,B 0,C 180,E1 -16335.046,E2 -16335.046} C_VEL
LIN {X 0,Y 298.45,Z 401.802,A -85,B 0,C 180,E1 -16338.749,E2 -16338.749} C_VEL
LIN {X 0,Y 298.468,Z 401.806,A -85,B 0,C 180,E1 -16343.186,E2 -16343.186} C_VEL
LIN {X 0,Y 298.393,Z 401.817,A -85,B 0,C 180,E1 -16347.199,E2 -16347.199} C_VEL
LIN {X 0,Y 298.429,Z 401.805,A -85,B 0,C 180,E1 -16350.614,E2 -16350.614} C_VEL
LIN {X 0,Y 298.481,Z 401.805,A -85,B 0,C 180,E1 -16353.474,E2 -16353.474} C_VEL
LIN {X 0,Y 298.428,Z 401.809,A -85,B 0,C 180,E1 -16356.699,E2 -16356.699} C_VEL
LIN {X 0,Y 298.522,Z 401.79,A -85,B 0,C 180,E1 -16360.756,E2 -16360.756} C_VEL
LIN {X 0,Y 298.59,Z 401.791,A -85,B 0,C 180,E1 -16364.994,E2 -16364.994} C_VEL
LIN {X 0,Y 298.587,Z 401.782,A -85,B 0,C 180,E1 -16369.146,E2 -16369.146} C_VEL
LIN {X 0,Y 298.737,Z 401.768,A -85,B 0,C 180,E1 -16371.885,E2 -16371.885} C_VEL
LIN {X 0,Y 298.653,Z 401.781,A -85,B 0,C 180,E1 -16374.599,E2 -16374.599} C_VEL
LIN {X 0,Y 298.919,Z 401.744,A -85,B 0,C 180,E1 -16378.653,E2 -16378.653} C_VEL
LIN {X 0,Y 298.919,Z 401.739,A -85,B 0,C 180,E1 -16381.347,E2 -16381.347} C_VEL
LIN {X 0,Y 298.784,Z 401.766,A -85,B 0,C 180,E1 -16386.754,E2 -16386.754} C_VEL
LIN {X 0,Y 298.631,Z 401.781,A -85,B 0,C 180,E1 -16389.482,E2 -16389.482} C_VEL
LIN {X 0,Y 298.547,Z 401.789,A -85,B 0,C 180,E1 -16393.616,E2 -16393.616} C_VEL
LIN {X 0,Y 298.545,Z 401.793,A -85,B 0,C 180,E1 -16396.409,E2 -16396.409} C_VEL
LIN {X 0,Y 298.508,Z 401.799,A -85,B 0,C 180,E1 -16399.655,E2 -16399.655} C_VEL
LIN {X 0,Y 298.454,Z 401.796,A -85,B 0,C 180,E1 -16403.598,E2 -16403.598} C_VEL
LIN {X 0,Y 298.486,Z 401.799,A -85,B 0,C 180,E1 -16406.575,E2 -16406.575} C_VEL
LIN {X 0,Y 298.418,Z 401.81,A -85,B 0,C 180,E1 -16409.641,E2 -16409.641} C_VEL
LIN {X 0,Y 298.393,Z 401.81,A -85,B 0,C 180,E1 -16412.8,E2 -16412.8} C_VEL
LIN {X 0,Y 298.442,Z 401.808,A -85,B 0,C 180,E1 -16416.807,E2 -16416.807} C_VEL
LIN {X 0,Y 298.385,Z 401.811,A -85,B 0,C 180,E1 -16421.088,E2 -16421.088} C_VEL
LIN {X 0,Y 298.387,Z 401.818,A -85,B 0,C 180,E1 -16425.042,E2 -16425.042} C_VEL
LIN {X 0,Y 298.417,Z 401.809,A -85,B 0,C 180,E1 -16428.906,E2 -16428.906} C_VEL
LIN {X 0,Y 298.465,Z 401.807,A -85,B 0,C 180,E1 -16433.188,E2 -16433.188} C_VEL
LIN {X 0,Y 298.395,Z 401.799,A -85,B 0,C 180,E1 -16437.2,E2 -16437.2} C_VEL
LIN {X 0,Y 298.432,Z 401.809,A -85,B 0,C 180,E1 -16440.615,E2 -16440.615} C_VEL
LIN {X 0,Y 298.477,Z 401.799,A -85,B 0,C 180,E1 -16443.477,E2 -16443.477} C_VEL
LIN {X 0,Y 298.435,Z 401.805,A -85,B 0,C 180,E1 -16446.698,E2 -16446.698} C_VEL
LIN {X 0,Y 298.54,Z 401.783,A -85,B 0,C 180,E1 -16450.757,E2 -16450.757} C_VEL
LIN {X 0,Y 298.608,Z 401.96,A -85,B 0,C 180,E1 -16454.473,E2 -16454.473} C_VEL
LIN {X 0,Y 300.545,Z 411.896,A -85,B 0,C 180,E1 -16457.851,E2 -16457.851} C_VEL
LIN {X 0,Y 300.886,Z 413.323,A -85,B 0,C 180,E1 -16458.035,E2 -16458.035} C_VEL
LIN {X 0,Y 304.349,Z 423.476,A -85,B 0,C 180,E1 -16458.547,E2 -16458.547} C_VEL
LIN {X 0,Y 307.475,Z 442.221,A -85,B 0,C 180,E1 -16459.222,E2 -16459.222} C_VEL
LIN {X 0,Y 308.18,Z 446.155,A -85,B 0,C 180,E1 -16459.365,E2 -16459.365} C_VEL
LIN {X 0,Y 306.458,Z 519.681,A -85,B 0,C 180,E1 -16461.087,E2 -16461.087} C_VEL
LIN {X 0,Y 305.847,Z 532.515,A -85,B 0,C 180,E1 -16461.638,E2 -16461.638} C_VEL
LIN {X 0,Y 304.897,Z 545.795,A -85,B 0,C 180,E1 -16462.488,E2 -16462.488} C_VEL
LIN {X 0,Y 303.726,Z 557.561,A -85,B 0,C 180,E1 -16463.523,E2 -16463.523} C_VEL
LIN {X 0,Y 302.368,Z 569.054,A -85,B 0,C 180,E1 -16464.832,E2 -16464.832} C_VEL
LIN {X 0,Y 301.056,Z 579.4,A -85,B 0,C 180,E1 -16466.319,E2 -16466.319} C_VEL
LIN {X 0,Y 299.88,Z 588.677,A -85,B 0,C 180,E1 -16467.985,E2 -16467.985} C_VEL
LIN {X 0,Y 298.912,Z 596.317,A -85,B 0,C 180,E1 -16469.663,E2 -16469.663} C_VEL
LIN {X 0,Y 297.994,Z 603.81,A -85,B 0,C 180,E1 -16471.689,E2 -16471.689} C_VEL
LIN {X 0,Y 297.181,Z 610.737,A -85,B 0,C 180,E1 -16474.068,E2 -16474.068} C_VEL
LIN {X 0,Y 296.896,Z 615.396,A -85,B 0,C 180,E1 -16476.17,E2 -16476.17} C_VEL
LIN {X 0,Y 296.522,Z 618.777,A -85,B 0,C 180,E1 -16478.175,E2 -16478.175} C_VEL
LIN {X 0,Y 296.373,Z 620.509,A -85,B 0,C 180,E1 -16479.554,E2 -16479.554} C_VEL
LIN {X 0,Y 296.294,Z 621.829,A -85,B 0,C 180,E1 -16480.938,E2 -16480.938} C_VEL
LIN {X 0,Y 296.317,Z 623.187,A -85,B 0,C 180,E1 -16483.485,E2 -16483.485} C_VEL
LIN {X 0,Y 296.283,Z 623.289,A -85,B 0,C 180,E1 -16485.124,E2 -16485.124} C_VEL
LIN {X 0,Y 296.35,Z 622.947,A -85,B 0,C 180,E1 -16486.533,E2 -16486.533} C_VEL
LIN {X 0,Y 296.754,Z 621.595,A -85,B 0,C 180,E1 -16488.681,E2 -16488.681} C_VEL
LIN {X 0,Y 297.417,Z 618.308,A -85,B 0,C 180,E1 -16491.485,E2 -16491.485} C_VEL
LIN {X 0,Y 298.243,Z 614.556,A -85,B 0,C 180,E1 -16493.615,E2 -16493.615} C_VEL
LIN {X 0,Y 299.387,Z 609.592,A -85,B 0,C 180,E1 -16495.739,E2 -16495.739} C_VEL
LIN {X 0,Y 300.851,Z 603.257,A -85,B 0,C 180,E1 -16497.852,E2 -16497.852} C_VEL
LIN {X 0,Y 302.651,Z 595.282,A -85,B 0,C 180,E1 -16499.95,E2 -16499.95} C_VEL
LIN {X 0,Y 304.525,Z 586.558,A -85,B 0,C 180,E1 -16501.766,E2 -16501.766} C_VEL
LIN {X 0,Y 306.552,Z 576.87,A -85,B 0,C 180,E1 -16503.381,E2 -16503.381} C_VEL
LIN {X 0,Y 308.38,Z 566.83,A -85,B 0,C 180,E1 -16504.732,E2 -16504.732} C_VEL
LIN {X 0,Y 310.086,Z 555.833,A -85,B 0,C 180,E1 -16505.906,E2 -16505.906} C_VEL
LIN {X 0,Y 311.637,Z 543.656,A -85,B 0,C 180,E1 -16506.9,E2 -16506.9} C_VEL
LIN {X 0,Y 312.971,Z 530.84,A -85,B 0,C 180,E1 -16507.653,E2 -16507.653} C_VEL
LIN {X 0,Y 313.774,Z 518.922,A -85,B 0,C 180,E1 -16508.12,E2 -16508.12} C_VEL
LIN {X 0,Y 315.876,Z 449.351,A -85,B 0,C 180,E1 -16509.751,E2 -16509.751} C_VEL
LIN {X 0,Y 313.668,Z 439.658,A -85,B 0,C 180,E1 -16510.255,E2 -16510.255} C_VEL
LIN {X 0,Y 306.607,Z 423.785,A -85,B 0,C 180,E1 -16511.514,E2 -16511.514} C_VEL
LIN {X 0,Y 301.181,Z 412.813,A -85,B 0,C 180,E1 -16512.547,E2 -16512.547} C_VEL
LIN {X 0,Y 300.519,Z 410.01,A -85,B 0,C 180,E1 -16513.533,E2 -16513.533} C_VEL
LIN {X 0,Y 298.534,Z 402.112,A -85,B 0,C 180,E1 -16516.826,E2 -16516.826} C_VEL
LIN {X 0,Y 297.906,Z 401.868,A -85,B 0,C 180,E1 -16517.532,E2 -16517.532} C_VEL
LIN {X 0,Y 294.477,Z 402.305,A -85,B 0,C 180,E1 -16519.72,E2 -16519.72} C_VEL
LIN {X 0,Y 292.259,Z 402.746,A -85,B 0,C 180,E1 -16521.241,E2 -16521.241} C_VEL
LIN {X 0,Y 291.429,Z 402.699,A -85,B 0,C 180,E1 -16522.419,E2 -16522.419} C_VEL
LIN {X 0,Y 291.411,Z 402.685,A -85,B 0,C 180,E1 -16522.816,E2 -16522.816} C_VEL
LIN {X 0,Y 291.34,Z 402.682,A -85,B 0,C 180,E1 -16526.301,E2 -16526.301} C_VEL
LIN {X 0,Y 291.382,Z 402.666,A -85,B 0,C 180,E1 -16530.259,E2 -16530.259} C_VEL
LIN {X 0,Y 291.414,Z 402.682,A -85,B 0,C 180,E1 -16534.272,E2 -16534.272} C_VEL
LIN {X 0,Y 291.376,Z 402.684,A -85,B 0,C 180,E1 -16537.299,E2 -16537.299} C_VEL
LIN {X 0,Y 291.456,Z 402.68,A -85,B 0,C 180,E1 -16540.27,E2 -16540.27} C_VEL
LIN {X 0,Y 291.534,Z 402.665,A -85,B 0,C 180,E1 -16544.634,E2 -16544.634} C_VEL
LIN {X 0,Y 291.531,Z 402.663,A -85,B 0,C 180,E1 -16548.881,E2 -16548.881} C_VEL
LIN {X 0,Y 291.702,Z 402.649,A -85,B 0,C 180,E1 -16551.688,E2 -16551.688} C_VEL
LIN {X 0,Y 291.627,Z 402.647,A -85,B 0,C 180,E1 -16554.468,E2 -16554.468} C_VEL
LIN {X 0,Y 291.888,Z 402.616,A -85,B 0,C 180,E1 -16558.62,E2 -16558.62} C_VEL
LIN {X 0,Y 291.886,Z 402.627,A -85,B 0,C 180,E1 -16561.38,E2 -16561.38} C_VEL
LIN {X 0,Y 291.739,Z 402.643,A -85,B 0,C 180,E1 -16566.918,E2 -16566.918} C_VEL
LIN {X 0,Y 291.623,Z 402.652,A -85,B 0,C 180,E1 -16569.712,E2 -16569.712} C_VEL
LIN {X 0,Y 291.516,Z 402.66,A -85,B 0,C 180,E1 -16573.951,E2 -16573.951} C_VEL
LIN {X 0,Y 291.48,Z 402.674,A -85,B 0,C 180,E1 -16576.818,E2 -16576.818} C_VEL
LIN {X 0,Y 291.445,Z 402.678,A -85,B 0,C 180,E1 -16579.875,E2 -16579.875} C_VEL
LIN {X 0,Y 291.394,Z 402.685,A -85,B 0,C 180,E1 -16584.206,E2 -16584.206} C_VEL
LIN {X 0,Y 291.417,Z 402.677,A -85,B 0,C 180,E1 -16587.272,E2 -16587.272} C_VEL
LIN {X 0,Y 291.332,Z 402.689,A -85,B 0,C 180,E1 -16590.438,E2 -16590.438} C_VEL
LIN {X 0,Y 291.34,Z 402.689,A -85,B 0,C 180,E1 -16593.699,E2 -16593.699} C_VEL
LIN {X 0,Y 291.4,Z 402.681,A -85,B 0,C 180,E1 -16597.262,E2 -16597.262} C_VEL
LIN {X 0,Y 291.401,Z 402.668,A -85,B 0,C 180,E1 -16600.631,E2 -16600.631} C_VEL
LIN {X 0,Y 291.35,Z 402.693,A -85,B 0,C 180,E1 -16604.391,E2 -16604.391} C_VEL
LIN {X 0,Y 291.349,Z 402.696,A -85,B 0,C 180,E1 -16608.4,E2 -16608.4} C_VEL
LIN {X 0,Y 291.362,Z 402.685,A -85,B 0,C 180,E1 -16611.161,E2 -16611.161} C_VEL
LIN {X 0,Y 291.424,Z 402.851,A -85,B 0,C 180,E1 -16613.14,E2 -16613.14} C_VEL
LIN {X 0,Y 293.216,Z 409.948,A -85,B 0,C 180,E1 -16616.134,E2 -16616.134} C_VEL
LIN {X 0,Y 295.389,Z 419.02,A -85,B 0,C 180,E1 -16619.63,E2 -16619.63} C_VEL
LIN {X 0,Y 295.915,Z 420.675,A -85,B 0,C 180,E1 -16619.888,E2 -16619.888} C_VEL
LIN {X 0,Y 302.008,Z 433.094,A -85,B 0,C 180,E1 -16621.033,E2 -16621.033} C_VEL
LIN {X 0,Y 305.394,Z 441.129,A -85,B 0,C 180,E1 -16621.672,E2 -16621.672} C_VEL
LIN {X 0,Y 309.273,Z 460.915,A -85,B 0,C 180,E1 -16622.67,E2 -16622.67} C_VEL
LIN {X 0,Y 309.497,Z 465,A -85,B 0,C 180,E1 -16622.806,E2 -16622.806} C_VEL
LIN {X 0,Y 307.353,Z 527.567,A -85,B 0,C 180,E1 -16624.296,E2 -16624.296} C_VEL
LIN {X 0,Y 306.325,Z 541.318,A -85,B 0,C 180,E1 -16624.885,E2 -16624.885} C_VEL
LIN {X 0,Y 304.814,Z 553.723,A -85,B 0,C 180,E1 -16625.662,E2 -16625.662} C_VEL
LIN {X 0,Y 303.238,Z 564.786,A -85,B 0,C 180,E1 -16626.617,E2 -16626.617} C_VEL
LIN {X 0,Y 301.231,Z 576.302,A -85,B 0,C 180,E1 -16627.902,E2 -16627.902} C_VEL
LIN {X 0,Y 299.187,Z 586.68,A -85,B 0,C 180,E1 -16629.369,E2 -16629.369} C_VEL
LIN {X 0,Y 297.205,Z 595.729,A -85,B 0,C 180,E1 -16630.958,E2 -16630.958} C_VEL
LIN {X 0,Y 295.178,Z 605.095,A -85,B 0,C 180,E1 -16633.043,E2 -16633.043} C_VEL
LIN {X 0,Y 293.351,Z 612.405,A -85,B 0,C 180,E1 -16635.076,E2 -16635.076} C_VEL
LIN {X 0,Y 292.158,Z 617.382,A -85,B 0,C 180,E1 -16636.79,E2 -16636.79} C_VEL
LIN {X 0,Y 291.079,Z 622.227,A -85,B 0,C 180,E1 -16638.864,E2 -16638.864} C_VEL
LIN {X 0,Y 290.253,Z 625.972,A -85,B 0,C 180,E1 -16640.945,E2 -16640.945} C_VEL
LIN {X 0,Y 289.719,Z 628.718,A -85,B 0,C 180,E1 -16643.034,E2 -16643.034} C_VEL
LIN {X 0,Y 289.557,Z 630.023,A -85,B 0,C 180,E1 -16644.429,E2 -16644.429} C_VEL
LIN {X 0,Y 289.421,Z 630.941,A -85,B 0,C 180,E1 -16645.823,E2 -16645.823} C_VEL
LIN {X 0,Y 289.396,Z 631.46,A -85,B 0,C 180,E1 -16647.216,E2 -16647.216} C_VEL
LIN {X 0,Y 289.373,Z 631.555,A -85,B 0,C 180,E1 -16648.609,E2 -16648.609} C_VEL
LIN {X 0,Y 289.382,Z 631.267,A -85,B 0,C 180,E1 -16650,E2 -16650} C_VEL
LIN {X 0,Y 289.373,Z 630.593,A -85,B 0,C 180,E1 -16651.392,E2 -16651.392} C_VEL
LIN {X 0,Y 289.392,Z 629.519,A -85,B 0,C 180,E1 -16652.784,E2 -16652.784} C_VEL
LIN {X 0,Y 289.428,Z 626.318,A -85,B 0,C 180,E1 -16655.388,E2 -16655.388} C_VEL
LIN {X 0,Y 289.731,Z 622.234,A -85,B 0,C 180,E1 -16657.667,E2 -16657.667} C_VEL
LIN {X 0,Y 290.223,Z 617.296,A -85,B 0,C 180,E1 -16659.76,E2 -16659.76} C_VEL
LIN {X 0,Y 290.928,Z 611.06,A -85,B 0,C 180,E1 -16661.849,E2 -16661.849} C_VEL
LIN {X 0,Y 292.001,Z 603.269,A -85,B 0,C 180,E1 -16663.927,E2 -16663.927} C_VEL
LIN {X 0,Y 293.091,Z 595.276,A -85,B 0,C 180,E1 -16665.65,E2 -16665.65} C_VEL
LIN {X 0,Y 294.343,Z 585.222,A -85,B 0,C 180,E1 -16667.411,E2 -16667.411} C_VEL
LIN {X 0,Y 295.631,Z 574.615,A -85,B 0,C 180,E1 -16668.899,E2 -16668.899} C_VEL
LIN {X 0,Y 296.913,Z 564.009,A -85,B 0,C 180,E1 -16670.073,E2 -16670.073} C_VEL
LIN {X 0,Y 298.138,Z 551.194,A -85,B 0,C 180,E1 -16671.159,E2 -16671.159} C_VEL
LIN {X 0,Y 299.073,Z 538.331,A -85,B 0,C 180,E1 -16671.949,E2 -16671.949} C_VEL
LIN {X 0,Y 299.766,Z 525.861,A -85,B 0,C 180,E1 -16672.44,E2 -16672.44} C_VEL
LIN {X 0,Y 301.13,Z 458.348,A -85,B 0,C 180,E1 -16674.058,E2 -16674.058} C_VEL
LIN {X 0,Y 295.905,Z 423.419,A -85,B 0,C 180,E1 -16675.315,E2 -16675.315} C_VEL
LIN {X 0,Y 294.818,Z 419.845,A -85,B 0,C 180,E1 -16675.532,E2 -16675.532} C_VEL
LIN {X 0,Y 292.943,Z 409.963,A -85,B 0,C 180,E1 -16678.673,E2 -16678.673} C_VEL
LIN {X 0,Y 291.401,Z 402.767,A -85,B 0,C 180,E1 -16681.183,E2 -16681.183} C_VEL
LIN {X 0,Y 291.386,Z 402.684,A -85,B 0,C 180,E1 -16685.37,E2 -16685.37} C_VEL
LIN {X 0,Y 291.365,Z 402.683,A -85,B 0,C 180,E1 -16688.839,E2 -16688.839} C_VEL
LIN {X 0,Y 291.348,Z 402.691,A -85,B 0,C 180,E1 -16692.487,E2 -16692.487} C_VEL
LIN {X 0,Y 291.369,Z 402.671,A -85,B 0,C 180,E1 -16696.353,E2 -16696.353} C_VEL
LIN {X 0,Y 291.405,Z 402.684,A -85,B 0,C 180,E1 -16700.512,E2 -16700.512} C_VEL
LIN {X 0,Y 291.432,Z 402.681,A -85,B 0,C 180,E1 -16702.923,E2 -16702.923} C_VEL
LIN {X 0,Y 291.343,Z 402.692,A -85,B 0,C 180,E1 -16706.301,E2 -16706.301} C_VEL
LIN {X 0,Y 291.385,Z 402.682,A -85,B 0,C 180,E1 -16710.26,E2 -16710.26} C_VEL
LIN {X 0,Y 291.413,Z 402.683,A -85,B 0,C 180,E1 -16714.271,E2 -16714.271} C_VEL
LIN {X 0,Y 291.371,Z 402.689,A -85,B 0,C 180,E1 -16717.298,E2 -16717.298} C_VEL
LIN {X 0,Y 291.455,Z 402.669,A -85,B 0,C 180,E1 -16720.27,E2 -16720.27} C_VEL
LIN {X 0,Y 291.537,Z 402.668,A -85,B 0,C 180,E1 -16724.634,E2 -16724.634} C_VEL
LIN {X 0,Y 291.531,Z 402.662,A -85,B 0,C 180,E1 -16728.88,E2 -16728.88} C_VEL
LIN {X 0,Y 291.684,Z 402.647,A -85,B 0,C 180,E1 -16731.688,E2 -16731.688} C_VEL
LIN {X 0,Y 291.624,Z 402.656,A -85,B 0,C 180,E1 -16734.468,E2 -16734.468} C_VEL
LIN {X 0,Y 291.886,Z 402.62,A -85,B 0,C 180,E1 -16738.62,E2 -16738.62} C_VEL
LIN {X 0,Y 291.886,Z 402.614,A -85,B 0,C 180,E1 -16741.38,E2 -16741.38} C_VEL
LIN {X 0,Y 291.732,Z 402.645,A -85,B 0,C 180,E1 -16746.918,E2 -16746.918} C_VEL
LIN {X 0,Y 291.571,Z 402.659,A -85,B 0,C 180,E1 -16749.714,E2 -16749.714} C_VEL
LIN {X 0,Y 291.517,Z 402.662,A -85,B 0,C 180,E1 -16753.95,E2 -16753.95} C_VEL
LIN {X 0,Y 291.483,Z 402.674,A -85,B 0,C 180,E1 -16756.818,E2 -16756.818} C_VEL
LIN {X 0,Y 291.448,Z 402.677,A -85,B 0,C 180,E1 -16759.875,E2 -16759.875} C_VEL
LIN {X 0,Y 291.397,Z 402.673,A -85,B 0,C 180,E1 -16764.205,E2 -16764.205} C_VEL
LIN {X 0,Y 291.42,Z 402.684,A -85,B 0,C 180,E1 -16767.272,E2 -16767.272} C_VEL
LIN {X 0,Y 291.335,Z 402.692,A -85,B 0,C 180,E1 -16770.437,E2 -16770.437} C_VEL
LIN {X 0,Y 291.342,Z 402.683,A -85,B 0,C 180,E1 -16773.699,E2 -16773.699} C_VEL
LIN {X 0,Y 291.37,Z 402.692,A -85,B 0,C 180,E1 -16777.253,E2 -16777.253} C_VEL
LIN {X 0,Y 291.33,Z 402.692,A -85,B 0,C 180,E1 -16780.643,E2 -16780.643} C_VEL
LIN {X 0,Y 291.312,Z 402.694,A -85,B 0,C 180,E1 -16784.398,E2 -16784.398} C_VEL
LIN {X 0,Y 291.354,Z 402.688,A -85,B 0,C 180,E1 -16788.398,E2 -16788.398} C_VEL
LIN {X 0,Y 291.374,Z 402.692,A -85,B 0,C 180,E1 -16791.162,E2 -16791.162} C_VEL
LIN {X 0,Y 291.385,Z 402.686,A -85,B 0,C 180,E1 -16794.63,E2 -16794.63} C_VEL
LIN {X 0,Y 291.371,Z 402.673,A -85,B 0,C 180,E1 -16797.951,E2 -16797.951} C_VEL
LIN {X 0,Y 291.382,Z 402.691,A -85,B 0,C 180,E1 -16801.159,E2 -16801.159} C_VEL
LIN {X 0,Y 291.413,Z 402.677,A -85,B 0,C 180,E1 -16804.272,E2 -16804.272} C_VEL
LIN {X 0,Y 291.382,Z 402.69,A -85,B 0,C 180,E1 -16807.3,E2 -16807.3} C_VEL
LIN {X 0,Y 291.459,Z 402.669,A -85,B 0,C 180,E1 -16810.27,E2 -16810.27} C_VEL
LIN {X 0,Y 291.555,Z 402.898,A -85,B 0,C 180,E1 -16814.14,E2 -16814.14} C_VEL
LIN {X 0,Y 293.398,Z 412.234,A -85,B 0,C 180,E1 -16817.374,E2 -16817.374} C_VEL
LIN {X 0,Y 294.118,Z 414.584,A -85,B 0,C 180,E1 -16817.581,E2 -16817.581} C_VEL
LIN {X 0,Y 297.953,Z 426.19,A -85,B 0,C 180,E1 -16818.161,E2 -16818.161} C_VEL
LIN {X 0,Y 301.483,Z 447.151,A -85,B 0,C 180,E1 -16818.939,E2 -16818.939} C_VEL
LIN {X 0,Y 299.718,Z 519.472,A -85,B 0,C 180,E1 -16820.664,E2 -16820.664} C_VEL
LIN {X 0,Y 299.074,Z 532.67,A -85,B 0,C 180,E1 -16821.242,E2 -16821.242} C_VEL
LIN {X 0,Y 298.191,Z 544.991,A -85,B 0,C 180,E1 -16822.041,E2 -16822.041} C_VEL
LIN {X 0,Y 297.037,Z 556.423,A -85,B 0,C 180,E1 -16823.035,E2 -16823.035} C_VEL
LIN {X 0,Y 295.642,Z 568.153,A -85,B 0,C 180,E1 -16824.372,E2 -16824.372} C_VEL
LIN {X 0,Y 294.225,Z 578.684,A -85,B 0,C 180,E1 -16825.89,E2 -16825.89} C_VEL
LIN {X 0,Y 292.979,Z 588.154,A -85,B 0,C 180,E1 -16827.594,E2 -16827.594} C_VEL
LIN {X 0,Y 291.998,Z 595.9,A -85,B 0,C 180,E1 -16829.31,E2 -16829.31} C_VEL
LIN {X 0,Y 290.999,Z 603.488,A -85,B 0,C 180,E1 -16831.384,E2 -16831.384} C_VEL
LIN {X 0,Y 290.216,Z 609.597,A -85,B 0,C 180,E1 -16833.47,E2 -16833.47} C_VEL
LIN {X 0,Y 289.849,Z 614.425,A -85,B 0,C 180,E1 -16835.565,E2 -16835.565} C_VEL
LIN {X 0,Y 289.507,Z 618.147,A -85,B 0,C 180,E1 -16837.672,E2 -16837.672} C_VEL
LIN {X 0,Y 289.267,Z 620.841,A -85,B 0,C 180,E1 -16839.791,E2 -16839.791} C_VEL
LIN {X 0,Y 289.184,Z 622.111,A -85,B 0,C 180,E1 -16841.21,E2 -16841.21} C_VEL
LIN {X 0,Y 289.216,Z 623.286,A -85,B 0,C 180,E1 -16843.589,E2 -16843.589} C_VEL
LIN {X 0,Y 289.209,Z 623.366,A -85,B 0,C 180,E1 -16845.503,E2 -16845.503} C_VEL
LIN {X 0,Y 289.326,Z 622.973,A -85,B 0,C 180,E1 -16846.947,E2 -16846.947} C_VEL
LIN {X 0,Y 289.694,Z 621.724,A -85,B 0,C 180,E1 -16848.89,E2 -16848.89} C_VEL
LIN {X 0,Y 290.256,Z 619.123,A -85,B 0,C 180,E1 -16851.296,E2 -16851.296} C_VEL
LIN {X 0,Y 291.052,Z 615.727,A -85,B 0,C 180,E1 -16853.425,E2 -16853.425} C_VEL
LIN {X 0,Y 292.234,Z 610.976,A -85,B 0,C 180,E1 -16855.65,E2 -16855.65} C_VEL
LIN {X 0,Y 293.858,Z 604.331,A -85,B 0,C 180,E1 -16858.008,E2 -16858.008} C_VEL
LIN {X 0,Y 295.478,Z 597.356,A -85,B 0,C 180,E1 -16859.965,E2 -16859.965} C_VEL
LIN {X 0,Y 297.502,Z 588.761,A -85,B 0,C 180,E1 -16861.896,E2 -16861.896} C_VEL
LIN {X 0,Y 299.661,Z 578.931,A -85,B 0,C 180,E1 -16863.646,E2 -16863.646} C_VEL
LIN {X 0,Y 301.8,Z 567.959,A -85,B 0,C 180,E1 -16865.193,E2 -16865.193} C_VEL
LIN {X 0,Y 303.586,Z 557.291,A -85,B 0,C 180,E1 -16866.384,E2 -16866.384} C_VEL
LIN {X 0,Y 305.151,Z 545.555,A -85,B 0,C 180,E1 -16867.404,E2 -16867.404} C_VEL
LIN {X 0,Y 306.651,Z 532.226,A -85,B 0,C 180,E1 -16868.227,E2 -16868.227} C_VEL
LIN {X 0,Y 307.581,Z 519.529,A -85,B 0,C 180,E1 -16868.753,E2 -16868.753} C_VEL
LIN {X 0,Y 309.821,Z 450.766,A -85,B 0,C 180,E1 -16870.393,E2 -16870.393} C_VEL
LIN {X 0,Y 307.969,Z 442.627,A -85,B 0,C 180,E1 -16870.831,E2 -16870.831} C_VEL
LIN {X 0,Y 301.445,Z 427.818,A -85,B 0,C 180,E1 -16872.037,E2 -16872.037} C_VEL
LIN {X 0,Y 294.089,Z 413.196,A -85,B 0,C 180,E1 -16873.458,E2 -16873.458} C_VEL
LIN {X 0,Y 293.846,Z 412.314,A -85,B 0,C 180,E1 -16873.657,E2 -16873.657} C_VEL
LIN {X 0,Y 291.9,Z 404.634,A -85,B 0,C 180,E1 -16876.883,E2 -16876.883} C_VEL
LIN {X 0,Y 291.427,Z 402.701,A -85,B 0,C 180,E1 -16877.864,E2 -16877.864} C_VEL
LIN {X 0,Y 291.38,Z 402.677,A -85,B 0,C 180,E1 -16881.163,E2 -16881.163} C_VEL
LIN {X 0,Y 291.411,Z 402.685,A -85,B 0,C 180,E1 -16882.816,E2 -16882.816} C_VEL
LIN {X 0,Y 290.86,Z 402.761,A -85,B 0,C 180,E1 -16883.969,E2 -16883.969} C_VEL
LIN {X 0,Y 289.297,Z 402.96,A -85,B 0,C 180,E1 -16885.099,E2 -16885.099} C_VEL
LIN {X 0,Y 285.474,Z 403.429,A -85,B 0,C 180,E1 -16887.366,E2 -16887.366} C_VEL
LIN {X 0,Y 284.379,Z 403.554,A -85,B 0,C 180,E1 -16888.548,E2 -16888.548} C_VEL
LIN {X 0,Y 284.287,Z 403.559,A -85,B 0,C 180,E1 -16888.949,E2 -16888.949} C_VEL
LIN {X 0,Y 284.394,Z 403.561,A -85,B 0,C 180,E1 -16892.825,E2 -16892.825} C_VEL
LIN {X 0,Y 284.361,Z 403.564,A -85,B 0,C 180,E1 -16896.707,E2 -16896.707} C_VEL
LIN {X 0,Y 284.399,Z 403.551,A -85,B 0,C 180,E1 -16901.261,E2 -16901.261} C_VEL
LIN {X 0,Y 284.471,Z 403.547,A -85,B 0,C 180,E1 -16904.469,E2 -16904.469} C_VEL
LIN {X 0,Y 284.483,Z 403.544,A -85,B 0,C 180,E1 -16908.601,E2 -16908.601} C_VEL
LIN {X 0,Y 284.652,Z 403.528,A -85,B 0,C 180,E1 -16911.481,E2 -16911.481} C_VEL
LIN {X 0,Y 284.597,Z 403.523,A -85,B 0,C 180,E1 -16914.331,E2 -16914.331} C_VEL
LIN {X 0,Y 284.854,Z 403.492,A -85,B 0,C 180,E1 -16918.586,E2 -16918.586} C_VEL
LIN {X 0,Y 284.852,Z 403.503,A -85,B 0,C 180,E1 -16921.414,E2 -16921.414} C_VEL
LIN {X 0,Y 284.691,Z 403.52,A -85,B 0,C 180,E1 -16927.09,E2 -16927.09} C_VEL
LIN {X 0,Y 284.56,Z 403.533,A -85,B 0,C 180,E1 -16929.956,E2 -16929.956} C_VEL
LIN {X 0,Y 284.476,Z 403.538,A -85,B 0,C 180,E1 -16934.303,E2 -16934.303} C_VEL
LIN {X 0,Y 284.419,Z 403.55,A -85,B 0,C 180,E1 -16937.249,E2 -16937.249} C_VEL
LIN {X 0,Y 284.373,Z 403.561,A -85,B 0,C 180,E1 -16940.243,E2 -16940.243} C_VEL
LIN {X 0,Y 284.363,Z 403.559,A -85,B 0,C 180,E1 -16943.876,E2 -16943.876} C_VEL
LIN {X 0,Y 284.392,Z 403.552,A -85,B 0,C 180,E1 -16947.174,E2 -16947.174} C_VEL
LIN {X 0,Y 284.29,Z 403.567,A -85,B 0,C 180,E1 -16951.275,E2 -16951.275} C_VEL
LIN {X 0,Y 284.358,Z 403.565,A -85,B 0,C 180,E1 -16955.355,E2 -16955.355} C_VEL
LIN {X 0,Y 284.334,Z 403.564,A -85,B 0,C 180,E1 -16958.166,E2 -16958.166} C_VEL
LIN {X 0,Y 284.338,Z 403.545,A -85,B 0,C 180,E1 -16962.142,E2 -16962.142} C_VEL
LIN {X 0,Y 284.294,Z 403.555,A -85,B 0,C 180,E1 -16966.198,E2 -16966.198} C_VEL
LIN {X 0,Y 284.31,Z 403.558,A -85,B 0,C 180,E1 -16970.023,E2 -16970.023} C_VEL
LIN {X 0,Y 284.352,Z 403.75,A -85,B 0,C 180,E1 -16972.271,E2 -16972.271} C_VEL
LIN {X 0,Y 286.335,Z 411.428,A -85,B 0,C 180,E1 -16975.632,E2 -16975.632} C_VEL
LIN {X 0,Y 288.249,Z 419.228,A -85,B 0,C 180,E1 -16978.714,E2 -16978.714} C_VEL
LIN {X 0,Y 290.184,Z 423.327,A -85,B 0,C 180,E1 -16979.192,E2 -16979.192} C_VEL
LIN {X 0,Y 297.554,Z 438.588,A -85,B 0,C 180,E1 -16980.627,E2 -16980.627} C_VEL
LIN {X 0,Y 299.83,Z 444.507,A -85,B 0,C 180,E1 -16981.085,E2 -16981.085} C_VEL
LIN {X 0,Y 303.366,Z 462.871,A -85,B 0,C 180,E1 -16982.035,E2 -16982.035} C_VEL
LIN {X 0,Y 302.964,Z 479.989,A -85,B 0,C 180,E1 -16982.464,E2 -16982.464} C_VEL
LIN {X 0,Y 301.205,Z 527.987,A -85,B 0,C 180,E1 -16983.635,E2 -16983.635} C_VEL
LIN {X 0,Y 300.137,Z 541.617,A -85,B 0,C 180,E1 -16984.237,E2 -16984.237} C_VEL
LIN {X 0,Y 298.569,Z 553.901,A -85,B 0,C 180,E1 -16985.025,E2 -16985.025} C_VEL
LIN {X 0,Y 296.788,Z 565.669,A -85,B 0,C 180,E1 -16986.077,E2 -16986.077} C_VEL
LIN {X 0,Y 294.716,Z 576.998,A -85,B 0,C 180,E1 -16987.386,E2 -16987.386} C_VEL
LIN {X 0,Y 292.598,Z 587.233,A -85,B 0,C 180,E1 -16988.883,E2 -16988.883} C_VEL
LIN {X 0,Y 290.471,Z 596.344,A -85,B 0,C 180,E1 -16990.544,E2 -16990.544} C_VEL
LIN {X 0,Y 288.408,Z 605.401,A -85,B 0,C 180,E1 -16992.633,E2 -16992.633} C_VEL
LIN {X 0,Y 286.508,Z 612.641,A -85,B 0,C 180,E1 -16994.711,E2 -16994.711} C_VEL
LIN {X 0,Y 285.223,Z 617.555,A -85,B 0,C 180,E1 -16996.463,E2 -16996.463} C_VEL
LIN {X 0,Y 284.086,Z 622.342,A -85,B 0,C 180,E1 -16998.586,E2 -16998.586} C_VEL
LIN {X 0,Y 283.244,Z 626.032,A -85,B 0,C 180,E1 -17000.719,E2 -17000.719} C_VEL
LIN {X 0,Y 282.669,Z 628.727,A -85,B 0,C 180,E1 -17002.859,E2 -17002.859} C_VEL
LIN {X 0,Y 282.473,Z 630.09,A -85,B 0,C 180,E1 -17004.393,E2 -17004.393} C_VEL
LIN {X 0,Y 282.307,Z 631.373,A -85,B 0,C 180,E1 -17007.146,E2 -17007.146} C_VEL
LIN {X 0,Y 282.298,Z 631.443,A -85,B 0,C 180,E1 -17008.574,E2 -17008.574} C_VEL
LIN {X 0,Y 282.304,Z 631.13,A -85,B 0,C 180,E1 -17010,E2 -17010} C_VEL
LIN {X 0,Y 282.298,Z 630.432,A -85,B 0,C 180,E1 -17011.427,E2 -17011.427} C_VEL
LIN {X 0,Y 282.301,Z 629.312,A -85,B 0,C 180,E1 -17012.854,E2 -17012.854} C_VEL
LIN {X 0,Y 282.336,Z 626.367,A -85,B 0,C 180,E1 -17015.316,E2 -17015.316} C_VEL
LIN {X 0,Y 282.687,Z 621.917,A -85,B 0,C 180,E1 -17017.859,E2 -17017.859} C_VEL
LIN {X 0,Y 283.197,Z 616.919,A -85,B 0,C 180,E1 -17020.004,E2 -17020.004} C_VEL
LIN {X 0,Y 283.925,Z 610.616,A -85,B 0,C 180,E1 -17022.146,E2 -17022.146} C_VEL
LIN {X 0,Y 285.091,Z 602.715,A -85,B 0,C 180,E1 -17024.272,E2 -17024.272} C_VEL
LIN {X 0,Y 286.235,Z 594.631,A -85,B 0,C 180,E1 -17026.035,E2 -17026.035} C_VEL
LIN {X 0,Y 287.56,Z 583.978,A -85,B 0,C 180,E1 -17027.917,E2 -17027.917} C_VEL
LIN {X 0,Y 288.847,Z 573.674,A -85,B 0,C 180,E1 -17029.361,E2 -17029.361} C_VEL
LIN {X 0,Y 290.151,Z 562.817,A -85,B 0,C 180,E1 -17030.562,E2 -17030.562} C_VEL
LIN {X 0,Y 291.502,Z 549.716,A -85,B 0,C 180,E1 -17031.665,E2 -17031.665} C_VEL
LIN {X 0,Y 292.424,Z 536.988,A -85,B 0,C 180,E1 -17032.429,E2 -17032.429} C_VEL
LIN {X 0,Y 293.084,Z 523.99,A -85,B 0,C 180,E1 -17032.922,E2 -17032.922} C_VEL
LIN {X 0,Y 294.455,Z 459.253,A -85,B 0,C 180,E1 -17034.5,E2 -17034.5} C_VEL
LIN {X 0,Y 289.491,Z 425.517,A -85,B 0,C 180,E1 -17035.746,E2 -17035.746} C_VEL
LIN {X 0,Y 287.543,Z 419.683,A -85,B 0,C 180,E1 -17036.1,E2 -17036.1} C_VEL
LIN {X 0,Y 285.878,Z 410.661,A -85,B 0,C 180,E1 -17039.05,E2 -17039.05} C_VEL
LIN {X 0,Y 284.367,Z 403.64,A -85,B 0,C 180,E1 -17041.576,E2 -17041.576} C_VEL
LIN {X 0,Y 284.362,Z 403.558,A -85,B 0,C 180,E1 -17045.353,E2 -17045.353} C_VEL
LIN {X 0,Y 284.323,Z 403.561,A -85,B 0,C 180,E1 -17048.167,E2 -17048.167} C_VEL
LIN {X 0,Y 284.296,Z 403.57,A -85,B 0,C 180,E1 -17052.13,E2 -17052.13} C_VEL
LIN {X 0,Y 284.317,Z 403.547,A -85,B 0,C 180,E1 -17056.201,E2 -17056.201} C_VEL
LIN {X 0,Y 284.35,Z 403.564,A -85,B 0,C 180,E1 -17060.013,E2 -17060.013} C_VEL
LIN {X 0,Y 284.354,Z 403.559,A -85,B 0,C 180,E1 -17063.617,E2 -17063.617} C_VEL
LIN {X 0,Y 284.306,Z 403.572,A -85,B 0,C 180,E1 -17067.189,E2 -17067.189} C_VEL
LIN {X 0,Y 284.356,Z 403.557,A -85,B 0,C 180,E1 -17070.376,E2 -17070.376} C_VEL
LIN {X 0,Y 284.375,Z 403.562,A -85,B 0,C 180,E1 -17073.586,E2 -17073.586} C_VEL
LIN {X 0,Y 284.33,Z 403.565,A -85,B 0,C 180,E1 -17076.704,E2 -17076.704} C_VEL
LIN {X 0,Y 284.396,Z 403.551,A -85,B 0,C 180,E1 -17081.261,E2 -17081.261} C_VEL
LIN {X 0,Y 284.475,Z 403.547,A -85,B 0,C 180,E1 -17084.469,E2 -17084.469} C_VEL
LIN {X 0,Y 284.484,Z 403.538,A -85,B 0,C 180,E1 -17088.601,E2 -17088.601} C_VEL
LIN {X 0,Y 284.635,Z 403.522,A -85,B 0,C 180,E1 -17091.48,E2 -17091.48} C_VEL
LIN {X 0,Y 284.594,Z 403.532,A -85,B 0,C 180,E1 -17094.331,E2 -17094.331} C_VEL
LIN {X 0,Y 284.852,Z 403.495,A -85,B 0,C 180,E1 -17098.586,E2 -17098.586} C_VEL
LIN {X 0,Y 284.852,Z 403.488,A -85,B 0,C 180,E1 -17101.414,E2 -17101.414} C_VEL
LIN {X 0,Y 284.683,Z 403.525,A -85,B 0,C 180,E1 -17107.09,E2 -17107.09} C_VEL
LIN {X 0,Y 284.515,Z 403.536,A -85,B 0,C 180,E1 -17109.957,E2 -17109.957} C_VEL
LIN {X 0,Y 284.474,Z 403.538,A -85,B 0,C 180,E1 -17114.303,E2 -17114.303} C_VEL
LIN {X 0,Y 284.422,Z 403.557,A -85,B 0,C 180,E1 -17117.248,E2 -17117.248} C_VEL
LIN {X 0,Y 284.376,Z 403.557,A -85,B 0,C 180,E1 -17120.242,E2 -17120.242} C_VEL
LIN {X 0,Y 284.365,Z 403.548,A -85,B 0,C 180,E1 -17123.875,E2 -17123.875} C_VEL
LIN {X 0,Y 284.394,Z 403.558,A -85,B 0,C 180,E1 -17127.174,E2 -17127.174} C_VEL
LIN {X 0,Y 284.293,Z 403.567,A -85,B 0,C 180,E1 -17131.275,E2 -17131.275} C_VEL
LIN {X 0,Y 284.338,Z 403.562,A -85,B 0,C 180,E1 -17135.348,E2 -17135.348} C_VEL
LIN {X 0,Y 284.306,Z 403.568,A -85,B 0,C 180,E1 -17138.17,E2 -17138.17} C_VEL
LIN {X 0,Y 284.267,Z 403.563,A -85,B 0,C 180,E1 -17142.125,E2 -17142.125} C_VEL
LIN {X 0,Y 284.285,Z 403.572,A -85,B 0,C 180,E1 -17146.196,E2 -17146.196} C_VEL
LIN {X 0,Y 284.35,Z 403.56,A -85,B 0,C 180,E1 -17150.013,E2 -17150.013} C_VEL
LIN {X 0,Y 284.351,Z 403.562,A -85,B 0,C 180,E1 -17153.617,E2 -17153.617} C_VEL
LIN {X 0,Y 284.307,Z 403.549,A -85,B 0,C 180,E1 -17157.19,E2 -17157.19} C_VEL
LIN {X 0,Y 284.359,Z 403.56,A -85,B 0,C 180,E1 -17160.376,E2 -17160.376} C_VEL
LIN {X 0,Y 284.375,Z 403.554,A -85,B 0,C 180,E1 -17163.587,E2 -17163.587} C_VEL
LIN {X 0,Y 284.367,Z 403.556,A -85,B 0,C 180,E1 -17166.707,E2 -17166.707} C_VEL
LIN {X 0,Y 284.403,Z 403.537,A -85,B 0,C 180,E1 -17171.262,E2 -17171.262} C_VEL
LIN {X 0,Y 284.468,Z 403.656,A -85,B 0,C 180,E1 -17173.678,E2 -17173.678} C_VEL
LIN {X 0,Y 286.187,Z 412.064,A -85,B 0,C 180,E1 -17176.744,E2 -17176.744} C_VEL
LIN {X 0,Y 286.415,Z 413.101,A -85,B 0,C 180,E1 -17176.922,E2 -17176.922} C_VEL
LIN {X 0,Y 291.317,Z 427.141,A -85,B 0,C 180,E1 -17177.693,E2 -17177.693} C_VEL
LIN {X 0,Y 294.784,Z 448.438,A -85,B 0,C 180,E1 -17178.5,E2 -17178.5} C_VEL
LIN {X 0,Y 292.997,Z 519.38,A -85,B 0,C 180,E1 -17180.227,E2 -17180.227} C_VEL
LIN {X 0,Y 292.344,Z 532.646,A -85,B 0,C 180,E1 -17180.818,E2 -17180.818} C_VEL
LIN {X 0,Y 291.352,Z 545.606,A -85,B 0,C 180,E1 -17181.678,E2 -17181.678} C_VEL
LIN {X 0,Y 290.206,Z 556.57,A -85,B 0,C 180,E1 -17182.66,E2 -17182.66} C_VEL
LIN {X 0,Y 288.734,Z 568.547,A -85,B 0,C 180,E1 -17184.062,E2 -17184.062} C_VEL
LIN {X 0,Y 287.28,Z 579.027,A -85,B 0,C 180,E1 -17185.615,E2 -17185.615} C_VEL
LIN {X 0,Y 286.124,Z 587.575,A -85,B 0,C 180,E1 -17187.184,E2 -17187.184} C_VEL
LIN {X 0,Y 285.108,Z 595.448,A -85,B 0,C 180,E1 -17188.94,E2 -17188.94} C_VEL
LIN {X 0,Y 283.999,Z 603.157,A -85,B 0,C 180,E1 -17191.063,E2 -17191.063} C_VEL
LIN {X 0,Y 283.345,Z 608.43,A -85,B 0,C 180,E1 -17192.843,E2 -17192.843} C_VEL
LIN {X 0,Y 282.866,Z 613.529,A -85,B 0,C 180,E1 -17194.988,E2 -17194.988} C_VEL
LIN {X 0,Y 282.5,Z 617.497,A -85,B 0,C 180,E1 -17197.145,E2 -17197.145} C_VEL
LIN {X 0,Y 282.274,Z 619.544,A -85,B 0,C 180,E1 -17198.591,E2 -17198.591} C_VEL
LIN {X 0,Y 282.139,Z 621.17,A -85,B 0,C 180,E1 -17200.041,E2 -17200.041} C_VEL
LIN {X 0,Y 282.089,Z 622.38,A -85,B 0,C 180,E1 -17201.496,E2 -17201.496} C_VEL
LIN {X 0,Y 282.121,Z 623.385,A -85,B 0,C 180,E1 -17203.702,E2 -17203.702} C_VEL
LIN {X 0,Y 282.133,Z 623.444,A -85,B 0,C 180,E1 -17205.902,E2 -17205.902} C_VEL
LIN {X 0,Y 282.3,Z 622.969,A -85,B 0,C 180,E1 -17207.382,E2 -17207.382} C_VEL
LIN {X 0,Y 282.644,Z 621.851,A -85,B 0,C 180,E1 -17209.112,E2 -17209.112} C_VEL
LIN {X 0,Y 283.343,Z 618.926,A -85,B 0,C 180,E1 -17211.842,E2 -17211.842} C_VEL
LIN {X 0,Y 284.32,Z 615.071,A -85,B 0,C 180,E1 -17214.199,E2 -17214.199} C_VEL
LIN {X 0,Y 285.5,Z 610.506,A -85,B 0,C 180,E1 -17216.301,E2 -17216.301} C_VEL
LIN {X 0,Y 287.189,Z 604.127,A -85,B 0,C 180,E1 -17218.575,E2 -17218.575} C_VEL
LIN {X 0,Y 289.061,Z 596.588,A -85,B 0,C 180,E1 -17220.701,E2 -17220.701} C_VEL
LIN {X 0,Y 290.959,Z 588.786,A -85,B 0,C 180,E1 -17222.467,E2 -17222.467} C_VEL
LIN {X 0,Y 293.28,Z 578.79,A -85,B 0,C 180,E1 -17224.272,E2 -17224.272} C_VEL
LIN {X 0,Y 295.37,Z 568.431,A -85,B 0,C 180,E1 -17225.764,E2 -17225.764} C_VEL
LIN {X 0,Y 297.381,Z 557.054,A -85,B 0,C 180,E1 -17227.058,E2 -17227.058} C_VEL
LIN {X 0,Y 299.023,Z 545.185,A -85,B 0,C 180,E1 -17228.093,E2 -17228.093} C_VEL
LIN {X 0,Y 300.571,Z 531.689,A -85,B 0,C 180,E1 -17228.93,E2 -17228.93} C_VEL
LIN {X 0,Y 301.514,Z 519.107,A -85,B 0,C 180,E1 -17229.447,E2 -17229.447} C_VEL
LIN {X 0,Y 303.799,Z 452.266,A -85,B 0,C 180,E1 -17231.059,E2 -17231.059} C_VEL
LIN {X 0,Y 302.298,Z 445.541,A -85,B 0,C 180,E1 -17231.43,E2 -17231.43} C_VEL
LIN {X 0,Y 296.082,Z 431.398,A -85,B 0,C 180,E1 -17232.622,E2 -17232.622} C_VEL
LIN {X 0,Y 288.504,Z 416.421,A -85,B 0,C 180,E1 -17234.11,E2 -17234.11} C_VEL
LIN {X 0,Y 286.749,Z 412.921,A -85,B 0,C 180,E1 -17234.538,E2 -17234.538} C_VEL
LIN {X 0,Y 284.837,Z 405.439,A -85,B 0,C 180,E1 -17237.748,E2 -17237.748} C_VEL
LIN {X 0,Y 284.37,Z 403.581,A -85,B 0,C 180,E1 -17238.734,E2 -17238.734} C_VEL
LIN {X 0,Y 284.325,Z 403.561,A -85,B 0,C 180,E1 -17242.815,E2 -17242.815} C_VEL
LIN {X 0,Y 284.318,Z 403.552,A -85,B 0,C 180,E1 -17245.352,E2 -17245.352} C_VEL
LIN {X 0,Y 284.287,Z 403.559,A -85,B 0,C 180,E1 -17248.949,E2 -17248.949} C_VEL
LIN {X 0,Y 283.615,Z 403.637,A -85,B 0,C 180,E1 -17250.133,E2 -17250.133} C_VEL
LIN {X 0,Y 280.778,Z 404.003,A -85,B 0,C 180,E1 -17252.062,E2 -17252.062} C_VEL
LIN {X 0,Y 278.384,Z 404.308,A -85,B 0,C 180,E1 -17253.629,E2 -17253.629} C_VEL
LIN {X 0,Y 277.369,Z 404.43,A -85,B 0,C 180,E1 -17254.842,E2 -17254.842} C_VEL
LIN {X 0,Y 277.293,Z 404.44,A -85,B 0,C 180,E1 -17255.253,E2 -17255.253} C_VEL
LIN {X 0,Y 277.339,Z 404.439,A -85,B 0,C 180,E1 -17259.65,E2 -17259.65} C_VEL
LIN {X 0,Y 277.429,Z 404.426,A -85,B 0,C 180,E1 -17264.283,E2 -17264.283} C_VEL
LIN {X 0,Y 277.429,Z 404.427,A -85,B 0,C 180,E1 -17268.308,E2 -17268.308} C_VEL
LIN {X 0,Y 277.609,Z 404.403,A -85,B 0,C 180,E1 -17271.263,E2 -17271.263} C_VEL
LIN {X 0,Y 277.567,Z 404.398,A -85,B 0,C 180,E1 -17274.187,E2 -17274.187} C_VEL
LIN {X 0,Y 277.82,Z 404.368,A -85,B 0,C 180,E1 -17278.551,E2 -17278.551} C_VEL
LIN {X 0,Y 277.818,Z 404.379,A -85,B 0,C 180,E1 -17281.45,E2 -17281.45} C_VEL
LIN {X 0,Y 277.646,Z 404.396,A -85,B 0,C 180,E1 -17287.271,E2 -17287.271} C_VEL
LIN {X 0,Y 277.501,Z 404.413,A -85,B 0,C 180,E1 -17290.212,E2 -17290.212} C_VEL
LIN {X 0,Y 277.429,Z 404.419,A -85,B 0,C 180,E1 -17294.675,E2 -17294.675} C_VEL
LIN {X 0,Y 277.339,Z 404.431,A -85,B 0,C 180,E1 -17299.234,E2 -17299.234} C_VEL
LIN {X 0,Y 277.314,Z 404.438,A -85,B 0,C 180,E1 -17304.171,E2 -17304.171} C_VEL
LIN {X 0,Y 277.321,Z 404.434,A -85,B 0,C 180,E1 -17307.506,E2 -17307.506} C_VEL
LIN {X 0,Y 277.267,Z 404.44,A -85,B 0,C 180,E1 -17310.482,E2 -17310.482} C_VEL
LIN {X 0,Y 277.25,Z 404.443,A -85,B 0,C 180,E1 -17313.896,E2 -17313.896} C_VEL
LIN {X 0,Y 277.286,Z 404.439,A -85,B 0,C 180,E1 -17317.467,E2 -17317.467} C_VEL
LIN {X 0,Y 277.261,Z 404.424,A -85,B 0,C 180,E1 -17321.228,E2 -17321.228} C_VEL
LIN {X 0,Y 277.24,Z 404.44,A -85,B 0,C 180,E1 -17325.219,E2 -17325.219} C_VEL
LIN {X 0,Y 277.232,Z 404.442,A -85,B 0,C 180,E1 -17329.51,E2 -17329.51} C_VEL
LIN {X 0,Y 277.276,Z 404.582,A -85,B 0,C 180,E1 -17331.299,E2 -17331.299} C_VEL
LIN {X 0,Y 279.217,Z 411.809,A -85,B 0,C 180,E1 -17334.627,E2 -17334.627} C_VEL
LIN {X 0,Y 281.023,Z 419.151,A -85,B 0,C 180,E1 -17337.646,E2 -17337.646} C_VEL
LIN {X 0,Y 285.139,Z 427.349,A -85,B 0,C 180,E1 -17338.587,E2 -17338.587} C_VEL
LIN {X 0,Y 292.26,Z 442.18,A -85,B 0,C 180,E1 -17340.038,E2 -17340.038} C_VEL
LIN {X 0,Y 294.231,Z 447.359,A -85,B 0,C 180,E1 -17340.452,E2 -17340.452} C_VEL
LIN {X 0,Y 297.437,Z 464.388,A -85,B 0,C 180,E1 -17341.354,E2 -17341.354} C_VEL
LIN {X 0,Y 295.187,Z 527.307,A -85,B 0,C 180,E1 -17342.909,E2 -17342.909} C_VEL
LIN {X 0,Y 294.124,Z 540.417,A -85,B 0,C 180,E1 -17343.48,E2 -17343.48} C_VEL
LIN {X 0,Y 292.535,Z 552.996,A -85,B 0,C 180,E1 -17344.283,E2 -17344.283} C_VEL
LIN {X 0,Y 290.642,Z 564.996,A -85,B 0,C 180,E1 -17345.348,E2 -17345.348} C_VEL
LIN {X 0,Y 288.478,Z 576.43,A -85,B 0,C 180,E1 -17346.68,E2 -17346.68} C_VEL
LIN {X 0,Y 286.233,Z 586.749,A -85,B 0,C 180,E1 -17348.201,E2 -17348.201} C_VEL
LIN {X 0,Y 284.185,Z 595.202,A -85,B 0,C 180,E1 -17349.744,E2 -17349.744} C_VEL
LIN {X 0,Y 281.977,Z 604.384,A -85,B 0,C 180,E1 -17351.848,E2 -17351.848} C_VEL
LIN {X 0,Y 279.982,Z 611.777,A -85,B 0,C 180,E1 -17353.972,E2 -17353.972} C_VEL
LIN {X 0,Y 278.308,Z 617.734,A -85,B 0,C 180,E1 -17356.12,E2 -17356.12} C_VEL
LIN {X 0,Y 277.107,Z 622.458,A -85,B 0,C 180,E1 -17358.294,E2 -17358.294} C_VEL
LIN {X 0,Y 276.217,Z 626.092,A -85,B 0,C 180,E1 -17360.481,E2 -17360.481} C_VEL
LIN {X 0,Y 275.613,Z 628.736,A -85,B 0,C 180,E1 -17362.676,E2 -17362.676} C_VEL
LIN {X 0,Y 275.35,Z 630.261,A -85,B 0,C 180,E1 -17364.523,E2 -17364.523} C_VEL
LIN {X 0,Y 275.221,Z 631.284,A -85,B 0,C 180,E1 -17367.073,E2 -17367.073} C_VEL
LIN {X 0,Y 275.224,Z 631.33,A -85,B 0,C 180,E1 -17368.537,E2 -17368.537} C_VEL
LIN {X 0,Y 275.229,Z 630.994,A -85,B 0,C 180,E1 -17370,E2 -17370} C_VEL
LIN {X 0,Y 275.224,Z 630.27,A -85,B 0,C 180,E1 -17371.464,E2 -17371.464} C_VEL
LIN {X 0,Y 275.213,Z 629.102,A -85,B 0,C 180,E1 -17372.928,E2 -17372.928} C_VEL
LIN {X 0,Y 275.236,Z 626.44,A -85,B 0,C 180,E1 -17375.223,E2 -17375.223} C_VEL
LIN {X 0,Y 275.497,Z 623.036,A -85,B 0,C 180,E1 -17377.328,E2 -17377.328} C_VEL
LIN {X 0,Y 275.964,Z 618.368,A -85,B 0,C 180,E1 -17379.529,E2 -17379.529} C_VEL
LIN {X 0,Y 276.789,Z 611.302,A -85,B 0,C 180,E1 -17382.092,E2 -17382.092} C_VEL
LIN {X 0,Y 277.938,Z 603.643,A -85,B 0,C 180,E1 -17384.273,E2 -17384.273} C_VEL
LIN {X 0,Y 279.098,Z 595.781,A -85,B 0,C 180,E1 -17386.081,E2 -17386.081} C_VEL
LIN {X 0,Y 280.351,Z 586.362,A -85,B 0,C 180,E1 -17387.846,E2 -17387.846} C_VEL
LIN {X 0,Y 281.782,Z 575.44,A -85,B 0,C 180,E1 -17389.487,E2 -17389.487} C_VEL
LIN {X 0,Y 283.133,Z 565.111,A -85,B 0,C 180,E1 -17390.715,E2 -17390.715} C_VEL
LIN {X 0,Y 284.431,Z 552.785,A -85,B 0,C 180,E1 -17391.85,E2 -17391.85} C_VEL
LIN {X 0,Y 285.497,Z 539.788,A -85,B 0,C 180,E1 -17392.717,E2 -17392.717} C_VEL
LIN {X 0,Y 286.283,Z 526.599,A -85,B 0,C 180,E1 -17393.295,E2 -17393.295} C_VEL
LIN {X 0,Y 287.798,Z 460.109,A -85,B 0,C 180,E1 -17394.962,E2 -17394.962} C_VEL
LIN {X 0,Y 283.12,Z 427.776,A -85,B 0,C 180,E1 -17396.184,E2 -17396.184} C_VEL
LIN {X 0,Y 280.391,Z 419.807,A -85,B 0,C 180,E1 -17396.652,E2 -17396.652} C_VEL
LIN {X 0,Y 279.454,Z 414.556,A -85,B 0,C 180,E1 -17398.331,E2 -17398.331} C_VEL
LIN {X 0,Y 277.311,Z 404.557,A -85,B 0,C 180,E1 -17401.958,E2 -17401.958} C_VEL
LIN {X 0,Y 277.325,Z 404.439,A -85,B 0,C 180,E1 -17405.811,E2 -17405.811} C_VEL
LIN {X 0,Y 277.254,Z 404.44,A -85,B 0,C 180,E1 -17409.324,E2 -17409.324} C_VEL
LIN {X 0,Y 277.239,Z 404.447,A -85,B 0,C 180,E1 -17413.192,E2 -17413.192} C_VEL
LIN {X 0,Y 277.27,Z 404.427,A -85,B 0,C 180,E1 -17417.312,E2 -17417.312} C_VEL
LIN {X 0,Y 277.267,Z 404.446,A -85,B 0,C 180,E1 -17420.677,E2 -17420.677} C_VEL
LIN {X 0,Y 277.304,Z 404.434,A -85,B 0,C 180,E1 -17424.344,E2 -17424.344} C_VEL
LIN {X 0,Y 277.243,Z 404.451,A -85,B 0,C 180,E1 -17427.836,E2 -17427.836} C_VEL
LIN {X 0,Y 277.269,Z 404.439,A -85,B 0,C 180,E1 -17431.21,E2 -17431.21} C_VEL
LIN {X 0,Y 277.307,Z 404.44,A -85,B 0,C 180,E1 -17434.479,E2 -17434.479} C_VEL
LIN {X 0,Y 277.265,Z 404.442,A -85,B 0,C 180,E1 -17437.653,E2 -17437.653} C_VEL
LIN {X 0,Y 277.339,Z 404.426,A -85,B 0,C 180,E1 -17440.766,E2 -17440.766} C_VEL
LIN {X 0,Y 277.425,Z 404.429,A -85,B 0,C 180,E1 -17445.325,E2 -17445.325} C_VEL
LIN {X 0,Y 277.458,Z 404.408,A -85,B 0,C 180,E1 -17449.787,E2 -17449.787} C_VEL
LIN {X 0,Y 277.637,Z 404.395,A -85,B 0,C 180,E1 -17452.729,E2 -17452.729} C_VEL
LIN {X 0,Y 277.818,Z 404.371,A -85,B 0,C 180,E1 -17458.55,E2 -17458.55} C_VEL
LIN {X 0,Y 277.818,Z 404.363,A -85,B 0,C 180,E1 -17461.449,E2 -17461.449} C_VEL
LIN {X 0,Y 277.637,Z 404.402,A -85,B 0,C 180,E1 -17467.271,E2 -17467.271} C_VEL
LIN {X 0,Y 277.457,Z 404.414,A -85,B 0,C 180,E1 -17470.213,E2 -17470.213} C_VEL
LIN {X 0,Y 277.424,Z 404.417,A -85,B 0,C 180,E1 -17474.675,E2 -17474.675} C_VEL
LIN {X 0,Y 277.342,Z 404.438,A -85,B 0,C 180,E1 -17479.234,E2 -17479.234} C_VEL
LIN {X 0,Y 277.316,Z 404.424,A -85,B 0,C 180,E1 -17484.17,E2 -17484.17} C_VEL
LIN {X 0,Y 277.323,Z 404.439,A -85,B 0,C 180,E1 -17487.505,E2 -17487.505} C_VEL
LIN {X 0,Y 277.27,Z 404.444,A -85,B 0,C 180,E1 -17490.482,E2 -17490.482} C_VEL
LIN {X 0,Y 277.244,Z 404.437,A -85,B 0,C 180,E1 -17493.896,E2 -17493.896} C_VEL
LIN {X 0,Y 277.263,Z 404.448,A -85,B 0,C 180,E1 -17497.47,E2 -17497.47} C_VEL
LIN {X 0,Y 277.207,Z 404.445,A -85,B 0,C 180,E1 -17501.237,E2 -17501.237} C_VEL
LIN {X 0,Y 277.221,Z 404.455,A -85,B 0,C 180,E1 -17505.222,E2 -17505.222} C_VEL
LIN {X 0,Y 277.286,Z 404.44,A -85,B 0,C 180,E1 -17509.497,E2 -17509.497} C_VEL
LIN {X 0,Y 277.285,Z 404.446,A -85,B 0,C 180,E1 -17512.534,E2 -17512.534} C_VEL
LIN {X 0,Y 277.254,Z 404.433,A -85,B 0,C 180,E1 -17516.106,E2 -17516.106} C_VEL
LIN {X 0,Y 277.261,Z 404.441,A -85,B 0,C 180,E1 -17519.539,E2 -17519.539} C_VEL
LIN {X 0,Y 277.357,Z 404.433,A -85,B 0,C 180,E1 -17522.864,E2 -17522.864} C_VEL
LIN {X 0,Y 277.329,Z 404.428,A -85,B 0,C 180,E1 -17526.08,E2 -17526.08} C_VEL
LIN {X 0,Y 277.345,Z 404.417,A -85,B 0,C 180,E1 -17530.766,E2 -17530.766} C_VEL
LIN {X 0,Y 277.454,Z 404.625,A -85,B 0,C 180,E1 -17533.349,E2 -17533.349} C_VEL
LIN {X 0,Y 279.06,Z 412.504,A -85,B 0,C 180,E1 -17536.24,E2 -17536.24} C_VEL
LIN {X 0,Y 280.283,Z 416.065,A -85,B 0,C 180,E1 -17536.519,E2 -17536.519} C_VEL
LIN {X 0,Y 284.89,Z 429.462,A -85,B 0,C 180,E1 -17537.256,E2 -17537.256} C_VEL
LIN {X 0,Y 288.101,Z 449.284,A -85,B 0,C 180,E1 -17538.03,E2 -17538.03} C_VEL
LIN {X 0,Y 286.288,Z 519.263,A -85,B 0,C 180,E1 -17539.77,E2 -17539.77} C_VEL
LIN {X 0,Y 285.62,Z 532.379,A -85,B 0,C 180,E1 -17540.359,E2 -17540.359} C_VEL
LIN {X 0,Y 284.602,Z 545.402,A -85,B 0,C 180,E1 -17541.236,E2 -17541.236} C_VEL
LIN {X 0,Y 283.366,Z 556.88,A -85,B 0,C 180,E1 -17542.285,E2 -17542.285} C_VEL
LIN {X 0,Y 281.835,Z 568.941,A -85,B 0,C 180,E1 -17543.736,E2 -17543.736} C_VEL
LIN {X 0,Y 280.343,Z 579.37,A -85,B 0,C 180,E1 -17545.326,E2 -17545.326} C_VEL
LIN {X 0,Y 279.042,Z 588.726,A -85,B 0,C 180,E1 -17547.112,E2 -17547.112} C_VEL
LIN {X 0,Y 277.968,Z 596.409,A -85,B 0,C 180,E1 -17548.913,E2 -17548.913} C_VEL
LIN {X 0,Y 276.901,Z 603.943,A -85,B 0,C 180,E1 -17551.09,E2 -17551.09} C_VEL
LIN {X 0,Y 275.993,Z 610.91,A -85,B 0,C 180,E1 -17553.65,E2 -17553.65} C_VEL
LIN {X 0,Y 275.637,Z 615.869,A -85,B 0,C 180,E1 -17556.068,E2 -17556.068} C_VEL
LIN {X 0,Y 275.144,Z 619.925,A -85,B 0,C 180,E1 -17558.815,E2 -17558.815} C_VEL
LIN {X 0,Y 275.017,Z 621.499,A -85,B 0,C 180,E1 -17560.304,E2 -17560.304} C_VEL
LIN {X 0,Y 275.004,Z 622.611,A -85,B 0,C 180,E1 -17561.797,E2 -17561.797} C_VEL
LIN {X 0,Y 275.022,Z 623.482,A -85,B 0,C 180,E1 -17563.817,E2 -17563.817} C_VEL
LIN {X 0,Y 275.075,Z 623.509,A -85,B 0,C 180,E1 -17566.322,E2 -17566.322} C_VEL
LIN {X 0,Y 275.296,Z 622.944,A -85,B 0,C 180,E1 -17567.838,E2 -17567.838} C_VEL
LIN {X 0,Y 275.586,Z 621.968,A -85,B 0,C 180,E1 -17569.361,E2 -17569.361} C_VEL
LIN {X 0,Y 275.955,Z 620.576,A -85,B 0,C 180,E1 -17570.888,E2 -17570.888} C_VEL
LIN {X 0,Y 276.768,Z 617.591,A -85,B 0,C 180,E1 -17573.177,E2 -17573.177} C_VEL
LIN {X 0,Y 277.884,Z 613.486,A -85,B 0,C 180,E1 -17575.463,E2 -17575.463} C_VEL
LIN {X 0,Y 279.639,Z 607.066,A -85,B 0,C 180,E1 -17578.113,E2 -17578.113} C_VEL
LIN {X 0,Y 281.546,Z 600.002,A -85,B 0,C 180,E1 -17580.362,E2 -17580.362} C_VEL
LIN {X 0,Y 283.42,Z 593.046,A -85,B 0,C 180,E1 -17582.133,E2 -17582.133} C_VEL
LIN {X 0,Y 285.673,Z 583.866,A -85,B 0,C 180,E1 -17584.033,E2 -17584.033} C_VEL
LIN {X 0,Y 287.926,Z 574.048,A -85,B 0,C 180,E1 -17585.644,E2 -17585.644} C_VEL
LIN {X 0,Y 290.016,Z 563.568,A -85,B 0,C 180,E1 -17587.022,E2 -17587.022} C_VEL
LIN {X 0,Y 291.764,Z 553.133,A -85,B 0,C 180,E1 -17588.114,E2 -17588.114} C_VEL
LIN {X 0,Y 293.41,Z 541.277,A -85,B 0,C 180,E1 -17589.068,E2 -17589.068} C_VEL
LIN {X 0,Y 294.776,Z 528.44,A -85,B 0,C 180,E1 -17589.791,E2 -17589.791} C_VEL
LIN {X 0,Y 295.655,Z 515.281,A -85,B 0,C 180,E1 -17590.261,E2 -17590.261} C_VEL
LIN {X 0,Y 297.803,Z 453.353,A -85,B 0,C 180,E1 -17591.766,E2 -17591.766} C_VEL
LIN {X 0,Y 296.513,Z 448.02,A -85,B 0,C 180,E1 -17592.084,E2 -17592.084} C_VEL
LIN {X 0,Y 290.517,Z 434.43,A -85,B 0,C 180,E1 -17593.28,E2 -17593.28} C_VEL
LIN {X 0,Y 283.395,Z 420.32,A -85,B 0,C 180,E1 -17594.745,E2 -17594.745} C_VEL
LIN {X 0,Y 279.66,Z 413.21,A -85,B 0,C 180,E1 -17595.595,E2 -17595.595} C_VEL
LIN {X 0,Y 278.655,Z 409.661,A -85,B 0,C 180,E1 -17597.081,E2 -17597.081} C_VEL
LIN {X 0,Y 277.299,Z 404.465,A -85,B 0,C 180,E1 -17599.654,E2 -17599.654} C_VEL
LIN {X 0,Y 277.321,Z 404.43,A -85,B 0,C 180,E1 -17604.187,E2 -17604.187} C_VEL
LIN {X 0,Y 277.241,Z 404.452,A -85,B 0,C 180,E1 -17607.836,E2 -17607.836} C_VEL
LIN {X 0,Y 277.267,Z 404.428,A -85,B 0,C 180,E1 -17611.21,E2 -17611.21} C_VEL
LIN {X 0,Y 277.31,Z 404.437,A -85,B 0,C 180,E1 -17614.479,E2 -17614.479} C_VEL
LIN {X 0,Y 277.293,Z 404.44,A -85,B 0,C 180,E1 -17615.253,E2 -17615.253} C_VEL
LIN {X 0,Y 276.634,Z 404.528,A -85,B 0,C 180,E1 -17616.467,E2 -17616.467} C_VEL
LIN {X 0,Y 273.765,Z 404.882,A -85,B 0,C 180,E1 -17618.443,E2 -17618.443} C_VEL
LIN {X 0,Y 271.346,Z 405.185,A -85,B 0,C 180,E1 -17620.05,E2 -17620.05} C_VEL
LIN {X 0,Y 270.342,Z 405.302,A -85,B 0,C 180,E1 -17621.295,E2 -17621.295} C_VEL
LIN {X 0,Y 270.279,Z 405.309,A -85,B 0,C 180,E1 -17621.717,E2 -17621.717} C_VEL
LIN {X 0,Y 270.39,Z 405.296,A -85,B 0,C 180,E1 -17624.935,E2 -17624.935} C_VEL
LIN {X 0,Y 270.436,Z 405.286,A -85,B 0,C 180,E1 -17629.519,E2 -17629.519} C_VEL
LIN {X 0,Y 270.604,Z 405.278,A -85,B 0,C 180,E1 -17632.539,E2 -17632.539} C_VEL
LIN {X 0,Y 270.786,Z 405.244,A -85,B 0,C 180,E1 -17638.513,E2 -17638.513} C_VEL
LIN {X 0,Y 270.784,Z 405.255,A -85,B 0,C 180,E1 -17641.487,E2 -17641.487} C_VEL
LIN {X 0,Y 270.604,Z 405.273,A -85,B 0,C 180,E1 -17647.462,E2 -17647.462} C_VEL
LIN {X 0,Y 270.436,Z 405.295,A -85,B 0,C 180,E1 -17650.481,E2 -17650.481} C_VEL
LIN {X 0,Y 270.397,Z 405.299,A -85,B 0,C 180,E1 -17655.065,E2 -17655.065} C_VEL
LIN {X 0,Y 270.296,Z 405.313,A -85,B 0,C 180,E1 -17659.756,E2 -17659.756} C_VEL
LIN {X 0,Y 270.269,Z 405.319,A -85,B 0,C 180,E1 -17664.586,E2 -17664.586} C_VEL
LIN {X 0,Y 270.267,Z 405.316,A -85,B 0,C 180,E1 -17667.909,E2 -17667.909} C_VEL
LIN {X 0,Y 270.18,Z 405.325,A -85,B 0,C 180,E1 -17671.349,E2 -17671.349} C_VEL
LIN {X 0,Y 270.211,Z 405.322,A -85,B 0,C 180,E1 -17674.904,E2 -17674.904} C_VEL
LIN {X 0,Y 270.249,Z 405.324,A -85,B 0,C 180,E1 -17678.726,E2 -17678.726} C_VEL
LIN {X 0,Y 270.22,Z 405.306,A -85,B 0,C 180,E1 -17682.549,E2 -17682.549} C_VEL
LIN {X 0,Y 270.189,Z 405.312,A -85,B 0,C 180,E1 -17686.746,E2 -17686.746} C_VEL
LIN {X 0,Y 270.219,Z 405.471,A -85,B 0,C 180,E1 -17690.297,E2 -17690.297} C_VEL
LIN {X 0,Y 272.365,Z 413.314,A -85,B 0,C 180,E1 -17694.055,E2 -17694.055} C_VEL
LIN {X 0,Y 273.75,Z 419.111,A -85,B 0,C 180,E1 -17696.502,E2 -17696.502} C_VEL
LIN {X 0,Y 280.645,Z 432.342,A -85,B 0,C 180,E1 -17698.069,E2 -17698.069} C_VEL
LIN {X 0,Y 287.326,Z 446.613,A -85,B 0,C 180,E1 -17699.493,E2 -17699.493} C_VEL
LIN {X 0,Y 288.807,Z 450.954,A -85,B 0,C 180,E1 -17699.83,E2 -17699.83} C_VEL
LIN {X 0,Y 291.467,Z 465.619,A -85,B 0,C 180,E1 -17700.624,E2 -17700.624} C_VEL
LIN {X 0,Y 289.137,Z 527.521,A -85,B 0,C 180,E1 -17702.181,E2 -17702.181} C_VEL
LIN {X 0,Y 288.027,Z 540.728,A -85,B 0,C 180,E1 -17702.775,E2 -17702.775} C_VEL
LIN {X 0,Y 286.367,Z 553.198,A -85,B 0,C 180,E1 -17703.589,E2 -17703.589} C_VEL
LIN {X 0,Y 284.522,Z 564.325,A -85,B 0,C 180,E1 -17704.585,E2 -17704.585} C_VEL
LIN {X 0,Y 282.299,Z 575.86,A -85,B 0,C 180,E1 -17705.943,E2 -17705.943} C_VEL
LIN {X 0,Y 279.918,Z 586.263,A -85,B 0,C 180,E1 -17707.488,E2 -17707.488} C_VEL
LIN {X 0,Y 277.557,Z 595.657,A -85,B 0,C 180,E1 -17709.239,E2 -17709.239} C_VEL
LIN {X 0,Y 275.231,Z 604.712,A -85,B 0,C 180,E1 -17711.387,E2 -17711.387} C_VEL
LIN {X 0,Y 273.168,Z 612.03,A -85,B 0,C 180,E1 -17713.561,E2 -17713.561} C_VEL
LIN {X 0,Y 271.411,Z 617.921,A -85,B 0,C 180,E1 -17715.76,E2 -17715.76} C_VEL
LIN {X 0,Y 270.146,Z 622.584,A -85,B 0,C 180,E1 -17717.988,E2 -17717.988} C_VEL
LIN {X 0,Y 269.209,Z 626.16,A -85,B 0,C 180,E1 -17720.231,E2 -17720.231} C_VEL
LIN {X 0,Y 268.552,Z 628.749,A -85,B 0,C 180,E1 -17722.482,E2 -17722.482} C_VEL
LIN {X 0,Y 268.231,Z 630.372,A -85,B 0,C 180,E1 -17724.655,E2 -17724.655} C_VEL
LIN {X 0,Y 268.118,Z 631.196,A -85,B 0,C 180,E1 -17726.995,E2 -17726.995} C_VEL
LIN {X 0,Y 268.13,Z 631.217,A -85,B 0,C 180,E1 -17728.498,E2 -17728.498} C_VEL
LIN {X 0,Y 268.155,Z 630.857,A -85,B 0,C 180,E1 -17730,E2 -17730} C_VEL
LIN {X 0,Y 268.13,Z 630.095,A -85,B 0,C 180,E1 -17731.502,E2 -17731.502} C_VEL
LIN {X 0,Y 268.127,Z 628.891,A -85,B 0,C 180,E1 -17733.005,E2 -17733.005} C_VEL
LIN {X 0,Y 268.132,Z 626.532,A -85,B 0,C 180,E1 -17735.112,E2 -17735.112} C_VEL
LIN {X 0,Y 268.422,Z 622.716,A -85,B 0,C 180,E1 -17737.523,E2 -17737.523} C_VEL
LIN {X 0,Y 268.947,Z 617.99,A -85,B 0,C 180,E1 -17739.78,E2 -17739.78} C_VEL
LIN {X 0,Y 269.807,Z 610.855,A -85,B 0,C 180,E1 -17742.41,E2 -17742.41} C_VEL
LIN {X 0,Y 271.039,Z 603.096,A -85,B 0,C 180,E1 -17744.644,E2 -17744.644} C_VEL
LIN {X 0,Y 272.257,Z 595.126,A -85,B 0,C 180,E1 -17746.496,E2 -17746.496} C_VEL
LIN {X 0,Y 273.559,Z 585.364,A -85,B 0,C 180,E1 -17748.344,E2 -17748.344} C_VEL
LIN {X 0,Y 275.023,Z 574.515,A -85,B 0,C 180,E1 -17749.986,E2 -17749.986} C_VEL
LIN {X 0,Y 276.399,Z 563.968,A -85,B 0,C 180,E1 -17751.244,E2 -17751.244} C_VEL
LIN {X 0,Y 277.842,Z 551.25,A -85,B 0,C 180,E1 -17752.396,E2 -17752.396} C_VEL
LIN {X 0,Y 278.852,Z 538.505,A -85,B 0,C 180,E1 -17753.24,E2 -17753.24} C_VEL
LIN {X 0,Y 279.617,Z 525.602,A -85,B 0,C 180,E1 -17753.79,E2 -17753.79} C_VEL
LIN {X 0,Y 281.2,Z 461.317,A -85,B 0,C 180,E1 -17755.428,E2 -17755.428} C_VEL
LIN {X 0,Y 276.677,Z 429.734,A -85,B 0,C 180,E1 -17756.655,E2 -17756.655} C_VEL
LIN {X 0,Y 273.235,Z 419.735,A -85,B 0,C 180,E1 -17757.262,E2 -17757.262} C_VEL
LIN {X 0,Y 272.669,Z 416.846,A -85,B 0,C 180,E1 -17758.149,E2 -17758.149} C_VEL
LIN {X 0,Y 270.594,Z 406.991,A -85,B 0,C 180,E1 -17761.731,E2 -17761.731} C_VEL
LIN {X 0,Y 270.234,Z 405.352,A -85,B 0,C 180,E1 -17762.466,E2 -17762.466} C_VEL
LIN {X 0,Y 270.239,Z 405.323,A -85,B 0,C 180,E1 -17766.737,E2 -17766.737} C_VEL
LIN {X 0,Y 270.216,Z 405.324,A -85,B 0,C 180,E1 -17771.039,E2 -17771.039} C_VEL
LIN {X 0,Y 270.193,Z 405.303,A -85,B 0,C 180,E1 -17775.388,E2 -17775.388} C_VEL
LIN {X 0,Y 270.245,Z 405.318,A -85,B 0,C 180,E1 -17779.447,E2 -17779.447} C_VEL
LIN {X 0,Y 270.256,Z 405.313,A -85,B 0,C 180,E1 -17783.721,E2 -17783.721} C_VEL
LIN {X 0,Y 270.203,Z 405.327,A -85,B 0,C 180,E1 -17786.892,E2 -17786.892} C_VEL
LIN {X 0,Y 270.195,Z 405.32,A -85,B 0,C 180,E1 -17790.382,E2 -17790.382} C_VEL
LIN {X 0,Y 270.259,Z 405.32,A -85,B 0,C 180,E1 -17793.763,E2 -17793.763} C_VEL
LIN {X 0,Y 270.208,Z 405.326,A -85,B 0,C 180,E1 -17797.036,E2 -17797.036} C_VEL
LIN {X 0,Y 270.297,Z 405.302,A -85,B 0,C 180,E1 -17800.244,E2 -17800.244} C_VEL
LIN {X 0,Y 270.393,Z 405.303,A -85,B 0,C 180,E1 -17804.935,E2 -17804.935} C_VEL
LIN {X 0,Y 270.41,Z 405.284,A -85,B 0,C 180,E1 -17809.518,E2 -17809.518} C_VEL
LIN {X 0,Y 270.595,Z 405.271,A -85,B 0,C 180,E1 -17812.538,E2 -17812.538} C_VEL
LIN {X 0,Y 270.783,Z 405.247,A -85,B 0,C 180,E1 -17818.513,E2 -17818.513} C_VEL
LIN {X 0,Y 270.784,Z 405.237,A -85,B 0,C 180,E1 -17821.487,E2 -17821.487} C_VEL
LIN {X 0,Y 270.595,Z 405.278,A -85,B 0,C 180,E1 -17827.461,E2 -17827.461} C_VEL
LIN {X 0,Y 270.409,Z 405.292,A -85,B 0,C 180,E1 -17830.482,E2 -17830.482} C_VEL
LIN {X 0,Y 270.393,Z 405.295,A -85,B 0,C 180,E1 -17835.065,E2 -17835.065} C_VEL
LIN {X 0,Y 270.299,Z 405.311,A -85,B 0,C 180,E1 -17839.756,E2 -17839.756} C_VEL
LIN {X 0,Y 270.271,Z 405.301,A -85,B 0,C 180,E1 -17844.586,E2 -17844.586} C_VEL
LIN {X 0,Y 270.27,Z 405.316,A -85,B 0,C 180,E1 -17847.909,E2 -17847.909} C_VEL
LIN {X 0,Y 270.182,Z 405.323,A -85,B 0,C 180,E1 -17851.348,E2 -17851.348} C_VEL
LIN {X 0,Y 270.199,Z 405.316,A -85,B 0,C 180,E1 -17854.906,E2 -17854.906} C_VEL
LIN {X 0,Y 270.196,Z 405.328,A -85,B 0,C 180,E1 -17858.711,E2 -17858.711} C_VEL
LIN {X 0,Y 270.17,Z 405.324,A -85,B 0,C 180,E1 -17863.251,E2 -17863.251} C_VEL
LIN {X 0,Y 270.193,Z 405.324,A -85,B 0,C 180,E1 -17867.446,E2 -17867.446} C_VEL
LIN {X 0,Y 270.244,Z 405.324,A -85,B 0,C 180,E1 -17871.381,E2 -17871.381} C_VEL
LIN {X 0,Y 270.215,Z 405.314,A -85,B 0,C 180,E1 -17875.097,E2 -17875.097} C_VEL
LIN {X 0,Y 270.2,Z 405.313,A -85,B 0,C 180,E1 -17879.131,E2 -17879.131} C_VEL
LIN {X 0,Y 270.265,Z 405.319,A -85,B 0,C 180,E1 -17882.146,E2 -17882.146} C_VEL
LIN {X 0,Y 270.277,Z 405.301,A -85,B 0,C 180,E1 -17885.519,E2 -17885.519} C_VEL
LIN {X 0,Y 270.302,Z 405.297,A -85,B 0,C 180,E1 -17890.245,E2 -17890.245} C_VEL
LIN {X 0,Y 270.384,Z 405.428,A -85,B 0,C 180,E1 -17892.9,E2 -17892.9} C_VEL
LIN {X 0,Y 271.887,Z 412.651,A -85,B 0,C 180,E1 -17895.63,E2 -17895.63} C_VEL
LIN {X 0,Y 273.414,Z 416.985,A -85,B 0,C 180,E1 -17895.963,E2 -17895.963} C_VEL
LIN {X 0,Y 278.372,Z 431.072,A -85,B 0,C 180,E1 -17896.774,E2 -17896.774} C_VEL
LIN {X 0,Y 281.449,Z 450.529,A -85,B 0,C 180,E1 -17897.553,E2 -17897.553} C_VEL
LIN {X 0,Y 279.597,Z 519.072,A -85,B 0,C 180,E1 -17899.293,E2 -17899.293} C_VEL
LIN {X 0,Y 278.888,Z 532.286,A -85,B 0,C 180,E1 -17899.893,E2 -17899.893} C_VEL
LIN {X 0,Y 277.874,Z 545.297,A -85,B 0,C 180,E1 -17900.786,E2 -17900.786} C_VEL
LIN {X 0,Y 276.475,Z 557.769,A -85,B 0,C 180,E1 -17901.963,E2 -17901.963} C_VEL
LIN {X 0,Y 274.948,Z 569.3,A -85,B 0,C 180,E1 -17903.395,E2 -17903.395} C_VEL
LIN {X 0,Y 273.413,Z 579.687,A -85,B 0,C 180,E1 -17905.023,E2 -17905.023} C_VEL
LIN {X 0,Y 272.177,Z 588.16,A -85,B 0,C 180,E1 -17906.669,E2 -17906.669} C_VEL
LIN {X 0,Y 271.088,Z 595.963,A -85,B 0,C 180,E1 -17908.514,E2 -17908.514} C_VEL
LIN {X 0,Y 269.913,Z 603.603,A -85,B 0,C 180,E1 -17910.746,E2 -17910.746} C_VEL
LIN {X 0,Y 269.067,Z 609.746,A -85,B 0,C 180,E1 -17912.994,E2 -17912.994} C_VEL
LIN {X 0,Y 268.581,Z 615.286,A -85,B 0,C 180,E1 -17915.61,E2 -17915.61} C_VEL
LIN {X 0,Y 268.24,Z 618.36,A -85,B 0,C 180,E1 -17917.527,E2 -17917.527} C_VEL
LIN {X 0,Y 268.033,Z 620.302,A -85,B 0,C 180,E1 -17919.051,E2 -17919.051} C_VEL
LIN {X 0,Y 267.902,Z 621.792,A -85,B 0,C 180,E1 -17920.581,E2 -17920.581} C_VEL
LIN {X 0,Y 267.894,Z 622.837,A -85,B 0,C 180,E1 -17922.114,E2 -17922.114} C_VEL
LIN {X 0,Y 267.935,Z 623.581,A -85,B 0,C 180,E1 -17923.947,E2 -17923.947} C_VEL
LIN {X 0,Y 268.02,Z 623.54,A -85,B 0,C 180,E1 -17926.764,E2 -17926.764} C_VEL
LIN {X 0,Y 268.556,Z 622.11,A -85,B 0,C 180,E1 -17929.592,E2 -17929.592} C_VEL
LIN {X 0,Y 269.041,Z 620.421,A -85,B 0,C 180,E1 -17931.451,E2 -17931.451} C_VEL
LIN {X 0,Y 269.889,Z 617.425,A -85,B 0,C 180,E1 -17933.741,E2 -17933.741} C_VEL
LIN {X 0,Y 271.161,Z 613.09,A -85,B 0,C 180,E1 -17936.142,E2 -17936.142} C_VEL
LIN {X 0,Y 272.708,Z 607.853,A -85,B 0,C 180,E1 -17938.364,E2 -17938.364} C_VEL
LIN {X 0,Y 274.759,Z 600.608,A -85,B 0,C 180,E1 -17940.768,E2 -17940.768} C_VEL
LIN {X 0,Y 276.981,Z 592.747,A -85,B 0,C 180,E1 -17942.823,E2 -17942.823} C_VEL
LIN {X 0,Y 279.278,Z 583.752,A -85,B 0,C 180,E1 -17944.704,E2 -17944.704} C_VEL
LIN {X 0,Y 281.651,Z 573.896,A -85,B 0,C 180,E1 -17946.343,E2 -17946.343} C_VEL
LIN {X 0,Y 283.791,Z 563.657,A -85,B 0,C 180,E1 -17947.708,E2 -17947.708} C_VEL
LIN {X 0,Y 285.669,Z 552.867,A -85,B 0,C 180,E1 -17948.853,E2 -17948.853} C_VEL
LIN {X 0,Y 287.215,Z 542.108,A -85,B 0,C 180,E1 -17949.736,E2 -17949.736} C_VEL
LIN {X 0,Y 288.637,Z 529.712,A -85,B 0,C 180,E1 -17950.469,E2 -17950.469} C_VEL
LIN {X 0,Y 289.616,Z 516.26,A -85,B 0,C 180,E1 -17950.974,E2 -17950.974} C_VEL
LIN {X 0,Y 291.761,Z 453.96,A -85,B 0,C 180,E1 -17952.532,E2 -17952.532} C_VEL
LIN {X 0,Y 290.531,Z 449.933,A -85,B 0,C 180,E1 -17952.817,E2 -17952.817} C_VEL
LIN {X 0,Y 284.411,Z 436.12,A -85,B 0,C 180,E1 -17954.099,E2 -17954.099} C_VEL
LIN {X 0,Y 276.856,Z 421.437,A -85,B 0,C 180,E1 -17955.726,E2 -17955.726} C_VEL
LIN {X 0,Y 272.411,Z 413.367,A -85,B 0,C 180,E1 -17956.774,E2 -17956.774} C_VEL
LIN {X 0,Y 271.742,Z 410.996,A -85,B 0,C 180,E1 -17957.745,E2 -17957.745} C_VEL
LIN {X 0,Y 270.228,Z 405.366,A -85,B 0,C 180,E1 -17960.617,E2 -17960.617} C_VEL
LIN {X 0,Y 270.253,Z 405.317,A -85,B 0,C 180,E1 -17963.721,E2 -17963.721} C_VEL
LIN {X 0,Y 270.2,Z 405.322,A -85,B 0,C 180,E1 -17966.892,E2 -17966.892} C_VEL
LIN {X 0,Y 270.192,Z 405.304,A -85,B 0,C 180,E1 -17970.382,E2 -17970.382} C_VEL
LIN {X 0,Y 270.26,Z 405.32,A -85,B 0,C 180,E1 -17973.764,E2 -17973.764} C_VEL
LIN {X 0,Y 270.228,Z 405.32,A -85,B 0,C 180,E1 -17977.038,E2 -17977.038} C_VEL
LIN {X 0,Y 270.296,Z 405.316,A -85,B 0,C 180,E1 -17980.244,E2 -17980.244} C_VEL
LIN {X 0,Y 270.279,Z 405.309,A -85,B 0,C 180,E1 -17981.717,E2 -17981.717} C_VEL
LIN {X 0,Y 269.662,Z 405.393,A -85,B 0,C 180,E1 -17982.962,E2 -17982.962} C_VEL
LIN {X 0,Y 266.839,Z 405.747,A -85,B 0,C 180,E1 -17984.991,E2 -17984.991} C_VEL
LIN {X 0,Y 264.423,Z 406.048,A -85,B 0,C 180,E1 -17986.64,E2 -17986.64} C_VEL
LIN {X 0,Y 263.398,Z 406.175,A -85,B 0,C 180,E1 -17987.919,E2 -17987.919} C_VEL
LIN {X 0,Y 263.323,Z 406.177,A -85,B 0,C 180,E1 -17988.352,E2 -17988.352} C_VEL
LIN {X 0,Y 263.553,Z 406.147,A -85,B 0,C 180,E1 -17990.793,E2 -17990.793} C_VEL
LIN {X 0,Y 263.51,Z 406.15,A -85,B 0,C 180,E1 -17993.876,E2 -17993.876} C_VEL
LIN {X 0,Y 263.752,Z 406.12,A -85,B 0,C 180,E1 -17998.473,E2 -17998.473} C_VEL
LIN {X 0,Y 263.748,Z 406.131,A -85,B 0,C 180,E1 -18001.527,E2 -18001.527} C_VEL
LIN {X 0,Y 263.566,Z 406.148,A -85,B 0,C 180,E1 -18007.662,E2 -18007.662} C_VEL
LIN {X 0,Y 263.368,Z 406.178,A -85,B 0,C 180,E1 -18010.766,E2 -18010.766} C_VEL
LIN {X 0,Y 263.345,Z 406.181,A -85,B 0,C 180,E1 -18015.479,E2 -18015.479} C_VEL
LIN {X 0,Y 263.258,Z 406.192,A -85,B 0,C 180,E1 -18020.307,E2 -18020.307} C_VEL
LIN {X 0,Y 263.203,Z 406.197,A -85,B 0,C 180,E1 -18025.292,E2 -18025.292} C_VEL
LIN {X 0,Y 263.175,Z 406.205,A -85,B 0,C 180,E1 -18028.73,E2 -18028.73} C_VEL
LIN {X 0,Y 263.129,Z 406.209,A -85,B 0,C 180,E1 -18032.289,E2 -18032.289} C_VEL
LIN {X 0,Y 263.186,Z 406.203,A -85,B 0,C 180,E1 -18035.978,E2 -18035.978} C_VEL
LIN {X 0,Y 263.188,Z 406.19,A -85,B 0,C 180,E1 -18039.858,E2 -18039.858} C_VEL
LIN {X 0,Y 263.142,Z 406.208,A -85,B 0,C 180,E1 -18043.98,E2 -18043.98} C_VEL
LIN {X 0,Y 263.145,Z 406.209,A -85,B 0,C 180,E1 -18048.402,E2 -18048.402} C_VEL
LIN {X 0,Y 263.188,Z 406.393,A -85,B 0,C 180,E1 -18049.25,E2 -18049.25} C_VEL
LIN {X 0,Y 265.546,Z 414.883,A -85,B 0,C 180,E1 -18053.481,E2 -18053.481} C_VEL
LIN {X 0,Y 266.553,Z 418.964,A -85,B 0,C 180,E1 -18055.254,E2 -18055.254} C_VEL
LIN {X 0,Y 268.77,Z 423.208,A -85,B 0,C 180,E1 -18055.839,E2 -18055.839} C_VEL
LIN {X 0,Y 275.72,Z 436.449,A -85,B 0,C 180,E1 -18057.434,E2 -18057.434} C_VEL
LIN {X 0,Y 282.038,Z 450.039,A -85,B 0,C 180,E1 -18058.837,E2 -18058.837} C_VEL
LIN {X 0,Y 283.269,Z 453.846,A -85,B 0,C 180,E1 -18059.135,E2 -18059.135} C_VEL
LIN {X 0,Y 285.604,Z 467.216,A -85,B 0,C 180,E1 -18059.876,E2 -18059.876} C_VEL
LIN {X 0,Y 283.168,Z 527.507,A -85,B 0,C 180,E1 -18061.412,E2 -18061.412} C_VEL
LIN {X 0,Y 281.98,Z 541.115,A -85,B 0,C 180,E1 -18062.04,E2 -18062.04} C_VEL
LIN {X 0,Y 280.261,Z 553.449,A -85,B 0,C 180,E1 -18062.867,E2 -18062.867} C_VEL
LIN {X 0,Y 278.18,Z 565.262,A -85,B 0,C 180,E1 -18063.963,E2 -18063.963} C_VEL
LIN {X 0,Y 275.881,Z 576.6,A -85,B 0,C 180,E1 -18065.346,E2 -18065.346} C_VEL
LIN {X 0,Y 273.417,Z 586.853,A -85,B 0,C 180,E1 -18066.922,E2 -18066.922} C_VEL
LIN {X 0,Y 270.943,Z 596.09,A -85,B 0,C 180,E1 -18068.707,E2 -18068.707} C_VEL
LIN {X 0,Y 268.517,Z 605.042,A -85,B 0,C 180,E1 -18070.904,E2 -18070.904} C_VEL
LIN {X 0,Y 266.372,Z 612.283,A -85,B 0,C 180,E1 -18073.129,E2 -18073.129} C_VEL
LIN {X 0,Y 264.532,Z 618.107,A -85,B 0,C 180,E1 -18075.382,E2 -18075.382} C_VEL
LIN {X 0,Y 263.2,Z 622.709,A -85,B 0,C 180,E1 -18077.666,E2 -18077.666} C_VEL
LIN {X 0,Y 262.186,Z 626.228,A -85,B 0,C 180,E1 -18079.966,E2 -18079.966} C_VEL
LIN {X 0,Y 261.517,Z 628.764,A -85,B 0,C 180,E1 -18082.278,E2 -18082.278} C_VEL
LIN {X 0,Y 261.124,Z 630.471,A -85,B 0,C 180,E1 -18084.77,E2 -18084.77} C_VEL
LIN {X 0,Y 261.019,Z 631.107,A -85,B 0,C 180,E1 -18086.914,E2 -18086.914} C_VEL
LIN {X 0,Y 261.038,Z 631.104,A -85,B 0,C 180,E1 -18088.458,E2 -18088.458} C_VEL
LIN {X 0,Y 261.082,Z 630.719,A -85,B 0,C 180,E1 -18090,E2 -18090} C_VEL
LIN {X 0,Y 261.038,Z 629.906,A -85,B 0,C 180,E1 -18091.543,E2 -18091.543} C_VEL
LIN {X 0,Y 261.025,Z 628.674,A -85,B 0,C 180,E1 -18093.087,E2 -18093.087} C_VEL
LIN {X 0,Y 261.031,Z 626.599,A -85,B 0,C 180,E1 -18095.002,E2 -18095.002} C_VEL
LIN {X 0,Y 261.358,Z 622.387,A -85,B 0,C 180,E1 -18097.727,E2 -18097.727} C_VEL
LIN {X 0,Y 261.907,Z 617.598,A -85,B 0,C 180,E1 -18100.045,E2 -18100.045} C_VEL
LIN {X 0,Y 262.659,Z 611.523,A -85,B 0,C 180,E1 -18102.36,E2 -18102.36} C_VEL
LIN {X 0,Y 263.883,Z 603.955,A -85,B 0,C 180,E1 -18104.656,E2 -18104.656} C_VEL
LIN {X 0,Y 265.119,Z 596.21,A -85,B 0,C 180,E1 -18106.557,E2 -18106.557} C_VEL
LIN {X 0,Y 266.462,Z 586.738,A -85,B 0,C 180,E1 -18108.452,E2 -18108.452} C_VEL
LIN {X 0,Y 267.965,Z 576.196,A -85,B 0,C 180,E1 -18110.135,E2 -18110.135} C_VEL
LIN {X 0,Y 269.535,Z 564.471,A -85,B 0,C 180,E1 -18111.611,E2 -18111.611} C_VEL
LIN {X 0,Y 270.99,Z 551.969,A -85,B 0,C 180,E1 -18112.792,E2 -18112.792} C_VEL
LIN {X 0,Y 272.128,Z 538.753,A -85,B 0,C 180,E1 -18113.698,E2 -18113.698} C_VEL
LIN {X 0,Y 272.934,Z 525.536,A -85,B 0,C 180,E1 -18114.28,E2 -18114.28} C_VEL
LIN {X 0,Y 274.566,Z 462.174,A -85,B 0,C 180,E1 -18115.931,E2 -18115.931} C_VEL
LIN {X 0,Y 270.259,Z 431.822,A -85,B 0,C 180,E1 -18117.145,E2 -18117.145} C_VEL
LIN {X 0,Y 265.981,Z 419.488,A -85,B 0,C 180,E1 -18117.932,E2 -18117.932} C_VEL
LIN {X 0,Y 264.829,Z 413.764,A -85,B 0,C 180,E1 -18119.932,E2 -18119.932} C_VEL
LIN {X 0,Y 263.202,Z 406.234,A -85,B 0,C 180,E1 -18122.903,E2 -18122.903} C_VEL
LIN {X 0,Y 263.203,Z 406.2,A -85,B 0,C 180,E1 -18126.769,E2 -18126.769} C_VEL
LIN {X 0,Y 263.132,Z 406.201,A -85,B 0,C 180,E1 -18129.867,E2 -18129.867} C_VEL
LIN {X 0,Y 263.139,Z 406.194,A -85,B 0,C 180,E1 -18133.98,E2 -18133.98} C_VEL
LIN {X 0,Y 263.173,Z 406.194,A -85,B 0,C 180,E1 -18138.394,E2 -18138.394} C_VEL
LIN {X 0,Y 263.188,Z 406.199,A -85,B 0,C 180,E1 -18142.108,E2 -18142.108} C_VEL
LIN {X 0,Y 263.183,Z 406.202,A -85,B 0,C 180,E1 -18145.89,E2 -18145.89} C_VEL
LIN {X 0,Y 263.139,Z 406.203,A -85,B 0,C 180,E1 -18149.505,E2 -18149.505} C_VEL
LIN {X 0,Y 263.189,Z 406.195,A -85,B 0,C 180,E1 -18153.002,E2 -18153.002} C_VEL
LIN {X 0,Y 263.152,Z 406.203,A -85,B 0,C 180,E1 -18156.384,E2 -18156.384} C_VEL
LIN {X 0,Y 263.26,Z 406.177,A -85,B 0,C 180,E1 -18159.693,E2 -18159.693} C_VEL
LIN {X 0,Y 263.342,Z 406.18,A -85,B 0,C 180,E1 -18164.521,E2 -18164.521} C_VEL
LIN {X 0,Y 263.352,Z 406.163,A -85,B 0,C 180,E1 -18169.233,E2 -18169.233} C_VEL
LIN {X 0,Y 263.555,Z 406.148,A -85,B 0,C 180,E1 -18172.338,E2 -18172.338} C_VEL
LIN {X 0,Y 263.748,Z 406.123,A -85,B 0,C 180,E1 -18178.473,E2 -18178.473} C_VEL
LIN {X 0,Y 263.748,Z 406.112,A -85,B 0,C 180,E1 -18181.527,E2 -18181.527} C_VEL
LIN {X 0,Y 263.555,Z 406.153,A -85,B 0,C 180,E1 -18187.662,E2 -18187.662} C_VEL
LIN {X 0,Y 263.352,Z 406.168,A -85,B 0,C 180,E1 -18190.766,E2 -18190.766} C_VEL
LIN {X 0,Y 263.342,Z 406.176,A -85,B 0,C 180,E1 -18195.478,E2 -18195.478} C_VEL
LIN {X 0,Y 263.261,Z 406.187,A -85,B 0,C 180,E1 -18200.307,E2 -18200.307} C_VEL
LIN {X 0,Y 263.206,Z 406.186,A -85,B 0,C 180,E1 -18205.291,E2 -18205.291} C_VEL
LIN {X 0,Y 263.177,Z 406.201,A -85,B 0,C 180,E1 -18208.73,E2 -18208.73} C_VEL
LIN {X 0,Y 263.13,Z 406.197,A -85,B 0,C 180,E1 -18212.289,E2 -18212.289} C_VEL
LIN {X 0,Y 263.179,Z 406.199,A -85,B 0,C 180,E1 -18216.763,E2 -18216.763} C_VEL
LIN {X 0,Y 263.123,Z 406.195,A -85,B 0,C 180,E1 -18221.594,E2 -18221.594} C_VEL
LIN {X 0,Y 263.132,Z 406.207,A -85,B 0,C 180,E1 -18226.018,E2 -18226.018} C_VEL
LIN {X 0,Y 263.153,Z 406.2,A -85,B 0,C 180,E1 -18230.137,E2 -18230.137} C_VEL
LIN {X 0,Y 263.188,Z 406.197,A -85,B 0,C 180,E1 -18234.023,E2 -18234.023} C_VEL
LIN {X 0,Y 263.133,Z 406.18,A -85,B 0,C 180,E1 -18237.712,E2 -18237.712} C_VEL
LIN {X 0,Y 263.201,Z 406.199,A -85,B 0,C 180,E1 -18241.783,E2 -18241.783} C_VEL
LIN {X 0,Y 263.226,Z 406.177,A -85,B 0,C 180,E1 -18245.201,E2 -18245.201} C_VEL
LIN {X 0,Y 263.264,Z 406.18,A -85,B 0,C 180,E1 -18249.694,E2 -18249.694} C_VEL
LIN {X 0,Y 263.295,Z 406.256,A -85,B 0,C 180,E1 -18252.425,E2 -18252.425} C_VEL
LIN {X 0,Y 264.706,Z 412.817,A -85,B 0,C 180,E1 -18254.999,E2 -18254.999} C_VEL
LIN {X 0,Y 267.803,Z 421.138,A -85,B 0,C 180,E1 -18255.584,E2 -18255.584} C_VEL
LIN {X 0,Y 272.018,Z 433.608,A -85,B 0,C 180,E1 -18256.308,E2 -18256.308} C_VEL
LIN {X 0,Y 274.843,Z 451.166,A -85,B 0,C 180,E1 -18257.039,E2 -18257.039} C_VEL
LIN {X 0,Y 272.886,Z 519.58,A -85,B 0,C 180,E1 -18258.816,E2 -18258.816} C_VEL
LIN {X 0,Y 272.15,Z 532.863,A -85,B 0,C 180,E1 -18259.444,E2 -18259.444} C_VEL
LIN {X 0,Y 271.094,Z 545.708,A -85,B 0,C 180,E1 -18260.354,E2 -18260.354} C_VEL
LIN {X 0,Y 269.851,Z 556.566,A -85,B 0,C 180,E1 -18261.387,E2 -18261.387} C_VEL
LIN {X 0,Y 268.213,Z 568.37,A -85,B 0,C 180,E1 -18262.85,E2 -18262.85} C_VEL
LIN {X 0,Y 266.721,Z 578.912,A -85,B 0,C 180,E1 -18264.519,E2 -18264.519} C_VEL
LIN {X 0,Y 265.344,Z 587.544,A -85,B 0,C 180,E1 -18266.203,E2 -18266.203} C_VEL
LIN {X 0,Y 264.206,Z 595.474,A -85,B 0,C 180,E1 -18268.094,E2 -18268.094} C_VEL
LIN {X 0,Y 262.947,Z 603.254,A -85,B 0,C 180,E1 -18270.382,E2 -18270.382} C_VEL
LIN {X 0,Y 262.245,Z 608.555,A -85,B 0,C 180,E1 -18272.303,E2 -18272.303} C_VEL
LIN {X 0,Y 261.643,Z 613.701,A -85,B 0,C 180,E1 -18274.622,E2 -18274.622} C_VEL
LIN {X 0,Y 261.25,Z 617.701,A -85,B 0,C 180,E1 -18276.953,E2 -18276.953} C_VEL
LIN {X 0,Y 260.897,Z 620.664,A -85,B 0,C 180,E1 -18279.301,E2 -18279.301} C_VEL
LIN {X 0,Y 260.789,Z 622.066,A -85,B 0,C 180,E1 -18280.873,E2 -18280.873} C_VEL
LIN {X 0,Y 260.786,Z 623.063,A -85,B 0,C 180,E1 -18282.45,E2 -18282.45} C_VEL
LIN {X 0,Y 260.833,Z 623.675,A -85,B 0,C 180,E1 -18284.07,E2 -18284.07} C_VEL
LIN {X 0,Y 260.85,Z 623.833,A -85,B 0,C 180,E1 -18285.629,E2 -18285.629} C_VEL
LIN {X 0,Y 260.974,Z 623.568,A -85,B 0,C 180,E1 -18287.23,E2 -18287.23} C_VEL
LIN {X 0,Y 261.497,Z 622.253,A -85,B 0,C 180,E1 -18289.837,E2 -18289.837} C_VEL
LIN {X 0,Y 262.431,Z 619.319,A -85,B 0,C 180,E1 -18292.849,E2 -18292.849} C_VEL
LIN {X 0,Y 263.539,Z 615.745,A -85,B 0,C 180,E1 -18295.256,E2 -18295.256} C_VEL
LIN {X 0,Y 265.024,Z 610.975,A -85,B 0,C 180,E1 -18297.649,E2 -18297.649} C_VEL
LIN {X 0,Y 266.947,Z 604.855,A -85,B 0,C 180,E1 -18300.013,E2 -18300.013} C_VEL
LIN {X 0,Y 269.214,Z 597.157,A -85,B 0,C 180,E1 -18302.354,E2 -18302.354} C_VEL
LIN {X 0,Y 271.627,Z 588.682,A -85,B 0,C 180,E1 -18304.393,E2 -18304.393} C_VEL
LIN {X 0,Y 274.341,Z 578.428,A -85,B 0,C 180,E1 -18306.327,E2 -18306.327} C_VEL
LIN {X 0,Y 276.596,Z 568.648,A -85,B 0,C 180,E1 -18307.802,E2 -18307.802} C_VEL
LIN {X 0,Y 278.703,Z 558.047,A -85,B 0,C 180,E1 -18309.08,E2 -18309.08} C_VEL
LIN {X 0,Y 280.546,Z 546.48,A -85,B 0,C 180,E1 -18310.169,E2 -18310.169} C_VEL
LIN {X 0,Y 282.263,Z 533.349,A -85,B 0,C 180,E1 -18311.047,E2 -18311.047} C_VEL
LIN {X 0,Y 283.398,Z 520.682,A -85,B 0,C 180,E1 -18311.616,E2 -18311.616} C_VEL
LIN {X 0,Y 285.943,Z 455.69,A -85,B 0,C 180,E1 -18313.278,E2 -18313.278} C_VEL
LIN {X 0,Y 282.53,Z 446.924,A -85,B 0,C 180,E1 -18314.04,E2 -18314.04} C_VEL
LIN {X 0,Y 275.178,Z 431.604,A -85,B 0,C 180,E1 -18315.663,E2 -18315.663} C_VEL
LIN {X 0,Y 269.344,Z 420.931,A -85,B 0,C 180,E1 -18316.991,E2 -18316.991} C_VEL
LIN {X 0,Y 265.141,Z 413.428,A -85,B 0,C 180,E1 -18318.053,E2 -18318.053} C_VEL
LIN {X 0,Y 264.353,Z 410.521,A -85,B 0,C 180,E1 -18319.357,E2 -18319.357} C_VEL
LIN {X 0,Y 263.178,Z 406.223,A -85,B 0,C 180,E1 -18321.716,E2 -18321.716} C_VEL
LIN {X 0,Y 263.179,Z 406.185,A -85,B 0,C 180,E1 -18325.89,E2 -18325.89} C_VEL
LIN {X 0,Y 263.136,Z 406.185,A -85,B 0,C 180,E1 -18329.505,E2 -18329.505} C_VEL
LIN {X 0,Y 263.189,Z 406.204,A -85,B 0,C 180,E1 -18333.002,E2 -18333.002} C_VEL
LIN {X 0,Y 263.18,Z 406.204,A -85,B 0,C 180,E1 -18336.387,E2 -18336.387} C_VEL
LIN {X 0,Y 263.258,Z 406.193,A -85,B 0,C 180,E1 -18339.693,E2 -18339.693} C_VEL
LIN {X 0,Y 263.339,Z 406.177,A -85,B 0,C 180,E1 -18344.521,E2 -18344.521} C_VEL
LIN {X 0,Y 263.323,Z 406.177,A -85,B 0,C 180,E1 -18348.352,E2 -18348.352} C_VEL
LIN {X 0,Y 262.689,Z 406.254,A -85,B 0,C 180,E1 -18349.631,E2 -18349.631} C_VEL
LIN {X 0,Y 259.891,Z 406.612,A -85,B 0,C 180,E1 -18351.716,E2 -18351.716} C_VEL
LIN {X 0,Y 257.49,Z 406.903,A -85,B 0,C 180,E1 -18353.412,E2 -18353.412} C_VEL
LIN {X 0,Y 256.441,Z 407.03,A -85,B 0,C 180,E1 -18354.726,E2 -18354.726} C_VEL
LIN {X 0,Y 256.347,Z 407.044,A -85,B 0,C 180,E1 -18355.171,E2 -18355.171} C_VEL
LIN {X 0,Y 256.716,Z 406.996,A -85,B 0,C 180,E1 -18358.431,E2 -18358.431} C_VEL
LIN {X 0,Y 256.711,Z 407.008,A -85,B 0,C 180,E1 -18361.569,E2 -18361.569} C_VEL
LIN {X 0,Y 256.534,Z 407.021,A -85,B 0,C 180,E1 -18367.873,E2 -18367.873} C_VEL
LIN {X 0,Y 256.304,Z 407.06,A -85,B 0,C 180,E1 -18371.066,E2 -18371.066} C_VEL
LIN {X 0,Y 256.294,Z 407.06,A -85,B 0,C 180,E1 -18375.915,E2 -18375.915} C_VEL
LIN {X 0,Y 256.161,Z 407.075,A -85,B 0,C 180,E1 -18380.896,E2 -18380.896} C_VEL
LIN {X 0,Y 256.183,Z 407.072,A -85,B 0,C 180,E1 -18385.139,E2 -18385.139} C_VEL
LIN {X 0,Y 256.109,Z 407.08,A -85,B 0,C 180,E1 -18389.6,E2 -18389.6} C_VEL
LIN {X 0,Y 256.081,Z 407.083,A -85,B 0,C 180,E1 -18393.291,E2 -18393.291} C_VEL
LIN {X 0,Y 256.137,Z 407.073,A -85,B 0,C 180,E1 -18397.28,E2 -18397.28} C_VEL
LIN {X 0,Y 256.108,Z 407.058,A -85,B 0,C 180,E1 -18401.193,E2 -18401.193} C_VEL
LIN {X 0,Y 256.07,Z 407.072,A -85,B 0,C 180,E1 -18405.528,E2 -18405.528} C_VEL
LIN {X 0,Y 256.129,Z 407.197,A -85,B 0,C 180,E1 -18408.027,E2 -18408.027} C_VEL
LIN {X 0,Y 258.239,Z 414.952,A -85,B 0,C 180,E1 -18412.115,E2 -18412.115} C_VEL
LIN {X 0,Y 259.342,Z 418.934,A -85,B 0,C 180,E1 -18413.928,E2 -18413.928} C_VEL
LIN {X 0,Y 267.554,Z 433.984,A -85,B 0,C 180,E1 -18415.998,E2 -18415.998} C_VEL
LIN {X 0,Y 274.948,Z 449.259,A -85,B 0,C 180,E1 -18417.73,E2 -18417.73} C_VEL
LIN {X 0,Y 277.621,Z 455.805,A -85,B 0,C 180,E1 -18418.356,E2 -18418.356} C_VEL
LIN {X 0,Y 279.731,Z 467.733,A -85,B 0,C 180,E1 -18419.051,E2 -18419.051} C_VEL
LIN {X 0,Y 277.274,Z 527.303,A -85,B 0,C 180,E1 -18420.603,E2 -18420.603} C_VEL
LIN {X 0,Y 276.042,Z 540.757,A -85,B 0,C 180,E1 -18421.227,E2 -18421.227} C_VEL
LIN {X 0,Y 274.206,Z 553.684,A -85,B 0,C 180,E1 -18422.112,E2 -18422.112} C_VEL
LIN {X 0,Y 272.178,Z 564.636,A -85,B 0,C 180,E1 -18423.137,E2 -18423.137} C_VEL
LIN {X 0,Y 269.779,Z 576.071,A -85,B 0,C 180,E1 -18424.544,E2 -18424.544} C_VEL
LIN {X 0,Y 267.213,Z 586.397,A -85,B 0,C 180,E1 -18426.149,E2 -18426.149} C_VEL
LIN {X 0,Y 264.857,Z 594.856,A -85,B 0,C 180,E1 -18427.783,E2 -18427.783} C_VEL
LIN {X 0,Y 262.64,Z 602.668,A -85,B 0,C 180,E1 -18429.644,E2 -18429.644} C_VEL
LIN {X 0,Y 260.36,Z 610.328,A -85,B 0,C 180,E1 -18431.916,E2 -18431.916} C_VEL
LIN {X 0,Y 258.24,Z 616.5,A -85,B 0,C 180,E1 -18434.209,E2 -18434.209} C_VEL
LIN {X 0,Y 256.682,Z 621.419,A -85,B 0,C 180,E1 -18436.543,E2 -18436.543} C_VEL
LIN {X 0,Y 255.494,Z 625.234,A -85,B 0,C 180,E1 -18438.899,E2 -18438.899} C_VEL
LIN {X 0,Y 254.458,Z 628.778,A -85,B 0,C 180,E1 -18442.063,E2 -18442.063} C_VEL
LIN {X 0,Y 254.022,Z 630.554,A -85,B 0,C 180,E1 -18444.882,E2 -18444.882} C_VEL
LIN {X 0,Y 253.923,Z 631.019,A -85,B 0,C 180,E1 -18446.827,E2 -18446.827} C_VEL
LIN {X 0,Y 253.947,Z 630.991,A -85,B 0,C 180,E1 -18448.415,E2 -18448.415} C_VEL
LIN {X 0,Y 253.989,Z 630.573,A -85,B 0,C 180,E1 -18450,E2 -18450} C_VEL
LIN {X 0,Y 253.948,Z 629.716,A -85,B 0,C 180,E1 -18451.586,E2 -18451.586} C_VEL
LIN {X 0,Y 253.927,Z 628.457,A -85,B 0,C 180,E1 -18453.174,E2 -18453.174} C_VEL
LIN {X 0,Y 253.953,Z 626.588,A -85,B 0,C 180,E1 -18454.941,E2 -18454.941} C_VEL
LIN {X 0,Y 254.165,Z 623.425,A -85,B 0,C 180,E1 -18457.148,E2 -18457.148} C_VEL
LIN {X 0,Y 254.664,Z 618.969,A -85,B 0,C 180,E1 -18459.531,E2 -18459.531} C_VEL
LIN {X 0,Y 255.426,Z 613.292,A -85,B 0,C 180,E1 -18461.909,E2 -18461.909} C_VEL
LIN {X 0,Y 256.506,Z 606.155,A -85,B 0,C 180,E1 -18464.276,E2 -18464.276} C_VEL
LIN {X 0,Y 257.975,Z 597.229,A -85,B 0,C 180,E1 -18466.622,E2 -18466.622} C_VEL
LIN {X 0,Y 259.438,Z 587.539,A -85,B 0,C 180,E1 -18468.665,E2 -18468.665} C_VEL
LIN {X 0,Y 261.07,Z 576.569,A -85,B 0,C 180,E1 -18470.485,E2 -18470.485} C_VEL
LIN {X 0,Y 262.696,Z 564.952,A -85,B 0,C 180,E1 -18471.996,E2 -18471.996} C_VEL
LIN {X 0,Y 264.194,Z 552.697,A -85,B 0,C 180,E1 -18473.206,E2 -18473.206} C_VEL
LIN {X 0,Y 265.41,Z 538.997,A -85,B 0,C 180,E1 -18474.18,E2 -18474.18} C_VEL
LIN {X 0,Y 266.23,Z 526.1,A -85,B 0,C 180,E1 -18474.776,E2 -18474.776} C_VEL
LIN {X 0,Y 267.846,Z 462.213,A -85,B 0,C 180,E1 -18476.491,E2 -18476.491} C_VEL
LIN {X 0,Y 263.79,Z 433.586,A -85,B 0,C 180,E1 -18477.675,E2 -18477.675} C_VEL
LIN {X 0,Y 258.775,Z 419.372,A -85,B 0,C 180,E1 -18478.617,E2 -18478.617} C_VEL
LIN {X 0,Y 257.248,Z 412.186,A -85,B 0,C 180,E1 -18481.27,E2 -18481.27} C_VEL
LIN {X 0,Y 256.146,Z 407.161,A -85,B 0,C 180,E1 -18483.336,E2 -18483.336} C_VEL
LIN {X 0,Y 256.13,Z 407.078,A -85,B 0,C 180,E1 -18487.275,E2 -18487.275} C_VEL
LIN {X 0,Y 256.081,Z 407.085,A -85,B 0,C 180,E1 -18491.198,E2 -18491.198} C_VEL
LIN {X 0,Y 256.075,Z 407.056,A -85,B 0,C 180,E1 -18495.526,E2 -18495.526} C_VEL
LIN {X 0,Y 256.103,Z 407.074,A -85,B 0,C 180,E1 -18498.806,E2 -18498.806} C_VEL
LIN {X 0,Y 256.155,Z 407.075,A -85,B 0,C 180,E1 -18502.871,E2 -18502.871} C_VEL
LIN {X 0,Y 256.084,Z 407.085,A -85,B 0,C 180,E1 -18506.709,E2 -18506.709} C_VEL
LIN {X 0,Y 256.125,Z 407.069,A -85,B 0,C 180,E1 -18511.409,E2 -18511.409} C_VEL
LIN {X 0,Y 256.14,Z 407.079,A -85,B 0,C 180,E1 -18515.696,E2 -18515.696} C_VEL
LIN {X 0,Y 256.16,Z 407.062,A -85,B 0,C 180,E1 -18519.104,E2 -18519.104} C_VEL
LIN {X 0,Y 256.292,Z 407.059,A -85,B 0,C 180,E1 -18524.084,E2 -18524.084} C_VEL
LIN {X 0,Y 256.29,Z 407.052,A -85,B 0,C 180,E1 -18527.327,E2 -18527.327} C_VEL
LIN {X 0,Y 256.512,Z 407.025,A -85,B 0,C 180,E1 -18532.126,E2 -18532.126} C_VEL
LIN {X 0,Y 256.495,Z 407.033,A -85,B 0,C 180,E1 -18536.858,E2 -18536.858} C_VEL
LIN {X 0,Y 256.762,Z 406.981,A -85,B 0,C 180,E1 -18540,E2 -18540} C_VEL
LIN {X 0,Y 256.495,Z 407.022,A -85,B 0,C 180,E1 -18543.141,E2 -18543.141} C_VEL
LIN {X 0,Y 256.512,Z 407.03,A -85,B 0,C 180,E1 -18547.874,E2 -18547.874} C_VEL
LIN {X 0,Y 256.29,Z 407.036,A -85,B 0,C 180,E1 -18552.672,E2 -18552.672} C_VEL
LIN {X 0,Y 256.276,Z 407.057,A -85,B 0,C 180,E1 -18556.299,E2 -18556.299} C_VEL
LIN {X 0,Y 256.155,Z 407.069,A -85,B 0,C 180,E1 -18561.12,E2 -18561.12} C_VEL
LIN {X 0,Y 256.186,Z 407.057,A -85,B 0,C 180,E1 -18565.139,E2 -18565.139} C_VEL
LIN {X 0,Y 256.112,Z 407.08,A -85,B 0,C 180,E1 -18569.6,E2 -18569.6} C_VEL
LIN {X 0,Y 256.066,Z 407.071,A -85,B 0,C 180,E1 -18573.293,E2 -18573.293} C_VEL
LIN {X 0,Y 256.112,Z 407.084,A -85,B 0,C 180,E1 -18577.271,E2 -18577.271} C_VEL
LIN {X 0,Y 256.053,Z 407.077,A -85,B 0,C 180,E1 -18581.204,E2 -18581.204} C_VEL
LIN {X 0,Y 256.065,Z 407.089,A -85,B 0,C 180,E1 -18585.529,E2 -18585.529} C_VEL
LIN {X 0,Y 256.082,Z 407.078,A -85,B 0,C 180,E1 -18588.802,E2 -18588.802} C_VEL
LIN {X 0,Y 256.154,Z 407.08,A -85,B 0,C 180,E1 -18592.872,E2 -18592.872} C_VEL
LIN {X 0,Y 256.085,Z 407.057,A -85,B 0,C 180,E1 -18596.71,E2 -18596.71} C_VEL
LIN {X 0,Y 256.138,Z 407.08,A -85,B 0,C 180,E1 -18601.405,E2 -18601.405} C_VEL
LIN {X 0,Y 256.168,Z 407.056,A -85,B 0,C 180,E1 -18605.699,E2 -18605.699} C_VEL
LIN {X 0,Y 256.168,Z 407.07,A -85,B 0,C 180,E1 -18609.105,E2 -18609.105} C_VEL
LIN {X 0,Y 256.237,Z 407.205,A -85,B 0,C 180,E1 -18612.027,E2 -18612.027} C_VEL
LIN {X 0,Y 257.48,Z 412.886,A -85,B 0,C 180,E1 -18614.302,E2 -18614.302} C_VEL
LIN {X 0,Y 260.597,Z 421.083,A -85,B 0,C 180,E1 -18614.914,E2 -18614.914} C_VEL
LIN {X 0,Y 265.662,Z 435.753,A -85,B 0,C 180,E1 -18615.812,E2 -18615.812} C_VEL
LIN {X 0,Y 268.268,Z 451.783,A -85,B 0,C 180,E1 -18616.502,E2 -18616.502} C_VEL
LIN {X 0,Y 266.246,Z 519.387,A -85,B 0,C 180,E1 -18618.292,E2 -18618.292} C_VEL
LIN {X 0,Y 265.481,Z 532.79,A -85,B 0,C 180,E1 -18618.935,E2 -18618.935} C_VEL
LIN {X 0,Y 264.331,Z 546.094,A -85,B 0,C 180,E1 -18619.898,E2 -18619.898} C_VEL
LIN {X 0,Y 263.043,Z 556.997,A -85,B 0,C 180,E1 -18620.969,E2 -18620.969} C_VEL
LIN {X 0,Y 261.354,Z 568.725,A -85,B 0,C 180,E1 -18622.467,E2 -18622.467} C_VEL
LIN {X 0,Y 259.813,Z 579.223,A -85,B 0,C 180,E1 -18624.178,E2 -18624.178} C_VEL
LIN {X 0,Y 258.252,Z 588.698,A -85,B 0,C 180,E1 -18626.099,E2 -18626.099} C_VEL
LIN {X 0,Y 257.09,Z 596.435,A -85,B 0,C 180,E1 -18628.041,E2 -18628.041} C_VEL
LIN {X 0,Y 255.838,Z 604.024,A -85,B 0,C 180,E1 -18630.393,E2 -18630.393} C_VEL
LIN {X 0,Y 255.104,Z 609.21,A -85,B 0,C 180,E1 -18632.368,E2 -18632.368} C_VEL
LIN {X 0,Y 254.531,Z 614.231,A -85,B 0,C 180,E1 -18634.751,E2 -18634.751} C_VEL
